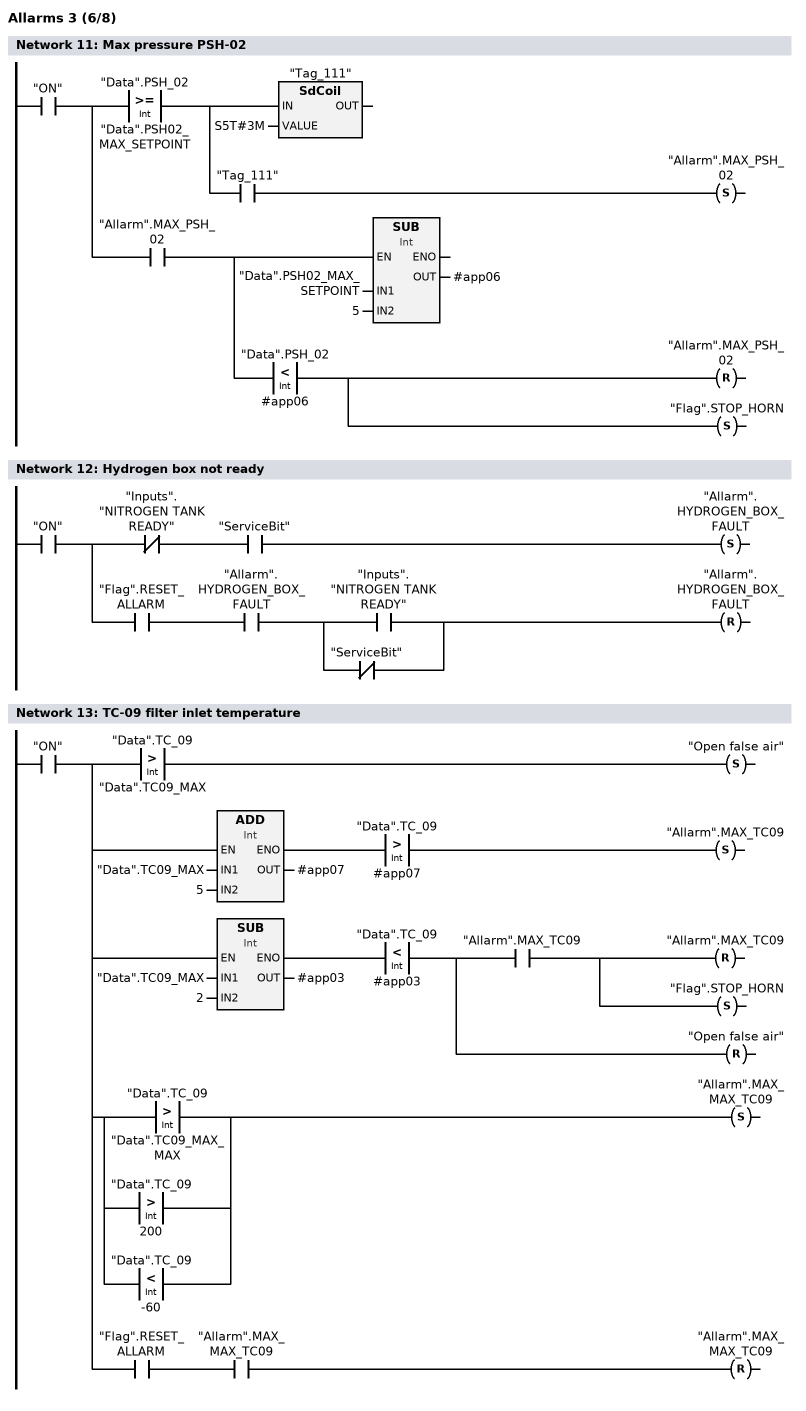
   // no SCL statement known for SdCoil: written as a call
   #_w1 := "ON" AND ("Data".PSH_02 >= "Data".PSH02_MAX_SETPOINT);
   #_w2 := "ON";
   SdCoil(in := #_w1, value := S5T#3M, operand := "Tag_111");
   IF #_w1 AND "Tag_111" THEN "Allarm".MAX_PSH_02 := TRUE; END_IF;
   #_w3 := #_w2 AND "Allarm".MAX_PSH_02;
   IF #_w3 THEN #app06 := "Data".PSH02_MAX_SETPOINT - 5; END_IF;
   IF #_w3 AND ("Data".PSH_02 < #app06) THEN
       "Allarm".MAX_PSH_02 := FALSE;
       "Flag".STOP_HORN := TRUE;
   END_IF;
END_REGION

REGION Network 12: Hydrogen box not ready
   RUNG wire#powerrail
      Contact( "ON" )
      wire#w1
      I_Contact( "Inputs"."NITROGEN TANK READY" )
      Contact( "ServiceBit" )
      S_Coil( "Allarm".HYDROGEN_BOX_FAULT )
   END_RUNG
   RUNG wire#w1
      Contact( "Flag".RESET_ALLARM )
      Contact( "Allarm".HYDROGEN_BOX_FAULT )
      wire#w2
      Contact( "Inputs"."NITROGEN TANK READY" )
      wire#w3
      R_Coil( "Allarm".HYDROGEN_BOX_FAULT )
   END_RUNG
   RUNG wire#w2
      I_Contact( "ServiceBit" )
   END_RUNG wire#w3
   // the same network as SCL:
   IF "ON" AND NOT "Inputs"."NITROGEN TANK READY" AND "ServiceBit" THEN
       "Allarm".HYDROGEN_BOX_FAULT := TRUE;
   END_IF;
   IF "ON" AND "Flag".RESET_ALLARM AND "Allarm".HYDROGEN_BOX_FAULT AND ("Inputs"."NITROGEN TANK READY" OR NOT "ServiceBit") THEN
       "Allarm".HYDROGEN_BOX_FAULT := FALSE;
   END_IF;
END_REGION

REGION Network 13: TC-09 filter inlet temperature
   RUNG wire#powerrail
      Contact( "ON" )
      wire#w1
      { S7_Templates := "SrcType := Int" } GT_Contact(in1 := "Data".TC_09, in2 := "Data".TC09_MAX)
      S_Coil( "Open false air" )
   END_RUNG
   RUNG wire#w1
      { S7_Templates := "SrcType := Int"; S7_GenerateENO := "TRUE" } Add(in1 := "Data".TC09_MAX, in2 := 5, out => #app07)
      { S7_Templates := "SrcType := Int" } GT_Contact(in1 := "Data".TC_09, in2 := #app07)
      S_Coil( "Allarm".MAX_TC09 )
   END_RUNG
   RUNG wire#w1
      { S7_Templates := "SrcType := Int"; S7_GenerateENO := "TRUE" } Sub(in1 := "Data".TC09_MAX, in2 := 2, out => #app03)
      { S7_Templates := "SrcType := Int" } LT_Contact(in1 := "Data".TC_09, in2 := #app03)
      wire#w2
      Contact( "Allarm".MAX_TC09 )
      wire#w3
      R_Coil( "Allarm".MAX_TC09 )
   END_RUNG
   RUNG wire#w3
      S_Coil( "Flag".STOP_HORN )
   END_RUNG
   RUNG wire#w2
      R_Coil( "Open false air" )
   END_RUNG
   RUNG wire#w1
      { S7_Templates := "SrcType := Int" } GT_Contact(in1 := "Data".TC_09, in2 := "Data".TC09_MAX_MAX)
      wire#w4
      S_Coil( "Allarm".MAX_MAX_TC09 )
   END_RUNG
   RUNG wire#w1
      { S7_Templates := "SrcType := Int" } GT_Contact(in1 := "Data".TC_09, in2 := 200)
   END_RUNG wire#w4
   RUNG wire#w1
      { S7_Templates := "SrcType := Int" } LT_Contact(in1 := "Data".TC_09, in2 := -60)
   END_RUNG wire#w4
   RUNG wire#w1
      Contact( "Flag".RESET_ALLARM )
      Contact( "Allarm".MAX_MAX_TC09 )
      R_Coil( "Allarm".MAX_MAX_TC09 )
   END_RUNG
   // the same network as SCL:
   // ENO of a box is taken as its EN; it also drops when the box reports an error
   IF "ON" AND ("Data".TC_09 > "Data".TC09_MAX) THEN "Open false air" := TRUE; END_IF;
   IF "ON" THEN #app07 := "Data".TC09_MAX + 5; END_IF;
   IF "ON" AND ("Data".TC_09 > #app07) THEN "Allarm".MAX_TC09 := TRUE; END_IF;
   IF "ON" THEN #app03 := "Data".TC09_MAX - 2; END_IF;
   #_w1 := "ON" AND ("Data".TC_09 < #app03);
   #_w2 := #_w1 AND "Allarm".MAX_TC09;
   IF #_w2 THEN
       "Allarm".MAX_TC09 := FALSE;
       "Flag".STOP_HORN := TRUE;
   END_IF;
   IF #_w1 THEN "Open false air" := FALSE; END_IF;
   IF "ON" AND (("Data".TC_09 > "Data".TC09_MAX_MAX) OR ("Data".TC_09 > 200) OR ("Data".TC_09 < (-60))) THEN
       "Allarm".MAX_MAX_TC09 := TRUE;
   END_IF;
   IF "ON" AND "Flag".RESET_ALLARM AND "Allarm".MAX_MAX_TC09 THEN "Allarm".MAX_MAX_TC09 := FALSE; END_IF;
END_REGION

REGION Network 14: Max filter depressure
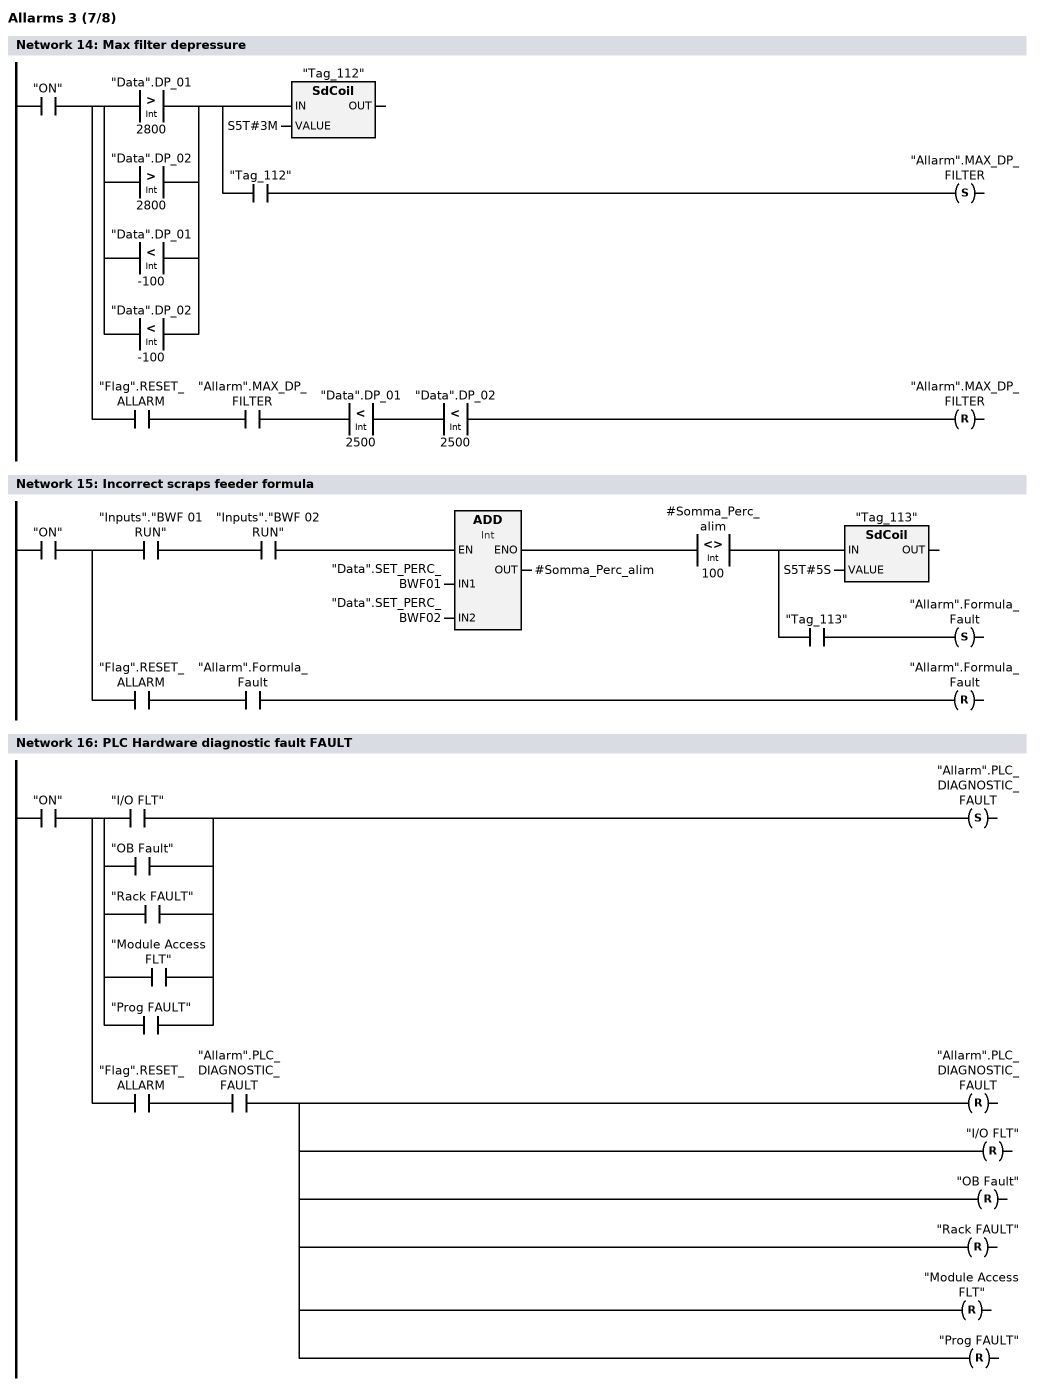
   // no SCL statement known for SdCoil: written as a call
   #_w1 := "ON" AND (("Data".DP_01 > 2800) OR ("Data".DP_02 > 2800) OR ("Data".DP_01 < (-100)) OR ("Data".DP_02 < (-100)));
   #_w2 := "ON";
   SdCoil(in := #_w1, value := S5T#3M, operand := "Tag_112");
   IF #_w1 AND "Tag_112" THEN "Allarm".MAX_DP_FILTER := TRUE; END_IF;
   IF #_w2 AND "Flag".RESET_ALLARM AND "Allarm".MAX_DP_FILTER AND ("Data".DP_01 < 2500) AND ("Data".DP_02 < 2500) THEN
       "Allarm".MAX_DP_FILTER := FALSE;
   END_IF;
END_REGION

REGION Network 15: Incorrect scraps feeder formula
   // no SCL statement known for SdCoil: written as a call
   // ENO of a box is taken as its EN; it also drops when the box reports an error
   #_w1 := "ON" AND "Inputs"."BWF 01 RUN" AND "Inputs"."BWF 02 RUN";
   IF #_w1 THEN #Somma_Perc_alim := "Data".SET_PERC_BWF01 + "Data".SET_PERC_BWF02; END_IF;
   #_w2 := #_w1 AND (#Somma_Perc_alim <> 100);
   #_w3 := "ON";
   SdCoil(in := #_w2, value := S5T#5S, operand := "Tag_113");
   IF #_w2 AND "Tag_113" THEN "Allarm".Formula_Fault := TRUE; END_IF;
   IF #_w3 AND "Flag".RESET_ALLARM AND "Allarm".Formula_Fault THEN "Allarm".Formula_Fault := FALSE; END_IF;
END_REGION

REGION Network 16: PLC Hardware diagnostic fault FAULT
   RUNG wire#powerrail
      Contact( "ON" )
      wire#w1
      Contact( "I/O FLT" )
      wire#w2
      S_Coil( "Allarm".PLC_DIAGNOSTIC_FAULT )
   END_RUNG
   RUNG wire#w1
      Contact( "OB Fault" )
   END_RUNG wire#w2
   RUNG wire#w1
      Contact( "Rack FAULT" )
   END_RUNG wire#w2
   RUNG wire#w1
      Contact( "Module Access FLT" )
   END_RUNG wire#w2
   RUNG wire#w1
      Contact( "Prog FAULT" )
   END_RUNG wire#w2
   RUNG wire#w1
      Contact( "Flag".RESET_ALLARM )
      Contact( "Allarm".PLC_DIAGNOSTIC_FAULT )
      wire#w3
      R_Coil( "Allarm".PLC_DIAGNOSTIC_FAULT )
   END_RUNG
   RUNG wire#w3
      R_Coil( "I/O FLT" )
   END_RUNG
   RUNG wire#w3
      R_Coil( "OB Fault" )
   END_RUNG
   RUNG wire#w3
      R_Coil( "Rack FAULT" )
   END_RUNG
   RUNG wire#w3
      R_Coil( "Module Access FLT" )
   END_RUNG
   RUNG wire#w3
      R_Coil( "Prog FAULT" )
   END_RUNG
   // the same network as SCL:
   IF "ON" AND ("I/O FLT" OR "OB Fault" OR "Rack FAULT" OR "Module Access FLT" OR "Prog FAULT") THEN
       "Allarm".PLC_DIAGNOSTIC_FAULT := TRUE;
   END_IF;
   #_w1 := "ON" AND "Flag".RESET_ALLARM AND "Allarm".PLC_DIAGNOSTIC_FAULT;
   IF #_w1 THEN
       "Allarm".PLC_DIAGNOSTIC_FAULT := FALSE;
       "I/O FLT" := FALSE;
       "OB Fault" := FALSE;
       "Rack FAULT" := FALSE;
       "Module Access FLT" := FALSE;
       "Prog FAULT" := FALSE;
   END_IF;
END_REGION

REGION Network 17: Ro03
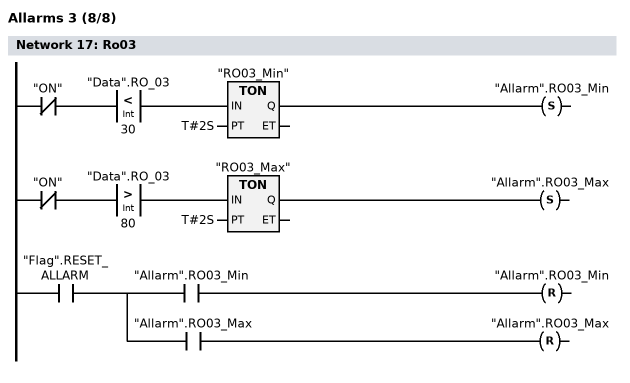
   "RO03_Min".TON(IN := NOT "ON" AND ("Data".RO_03 < 30), PT := T#2S);
   IF "RO03_Min".Q THEN "Allarm".RO03_Min := TRUE; END_IF;
   "RO03_Max".TON(IN := NOT "ON" AND ("Data".RO_03 > 80), PT := T#2S);
   IF "RO03_Max".Q THEN "Allarm".RO03_Max := TRUE; END_IF;
   IF "Flag".RESET_ALLARM AND "Allarm".RO03_Min THEN "Allarm".RO03_Min := FALSE; END_IF;
   IF "Flag".RESET_ALLARM AND "Allarm".RO03_Max THEN "Allarm".RO03_Max := FALSE; END_IF;
END_REGION
END_FUNCTION

FUNCTION "Motors 1" : Void   // FC7, LAD
{ S7_Optimized_Access := 'FALSE' }
VERSION : 0.1
   VAR_TEMP
      Start_LD01Vib : Bool;
      Disable_Load_RD01 : Bool;
      Stop_Fan_FN01 : Bool;
      Stop_Fan_FN04 : Bool;
      TimConv : Word;
   END_VAR
   VAR_TEMP   // added for the SCL form of the ladder/FBD networks
      _w1 : Bool;
      _w2 : Bool;
      _w3 : Bool;
   END_VAR
BEGIN

REGION Network 1: Enable maintenance mode / MAINTENANCE
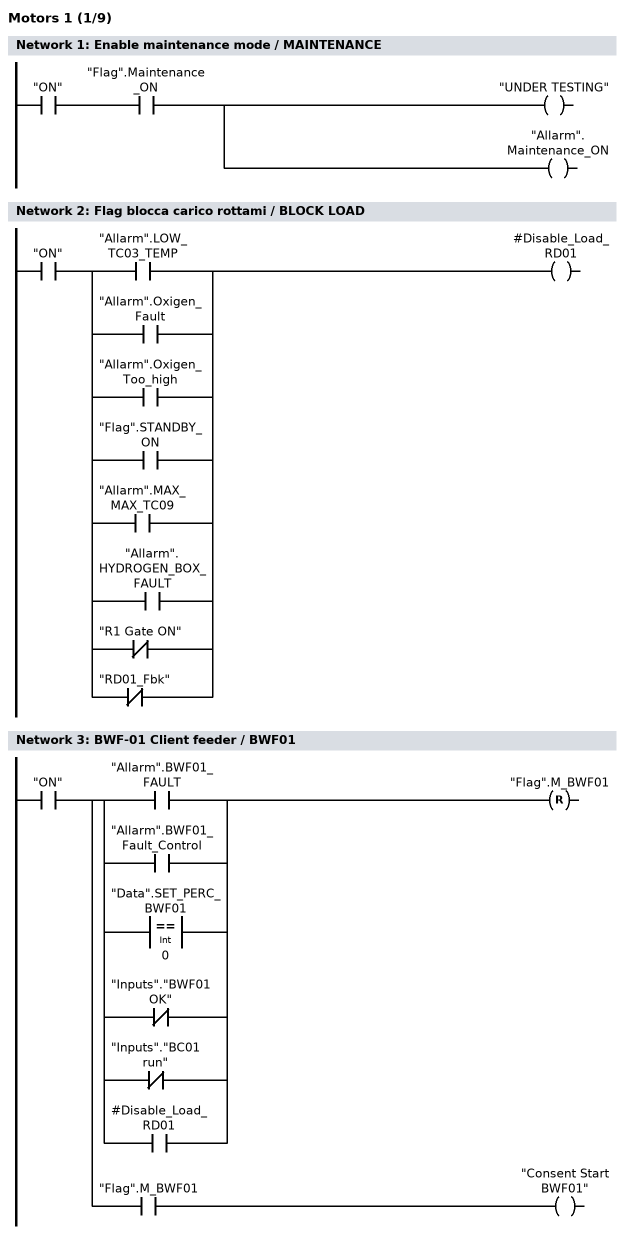
   RUNG wire#powerrail
      Contact( "ON" )
      Contact( "Flag".Maintenance_ON )
      wire#w1
      Coil( "UNDER TESTING" )
   END_RUNG
   RUNG wire#w1
      Coil( "Allarm".Maintenance_ON )
   END_RUNG
   // the same network as SCL:
   "UNDER TESTING" := "ON" AND "Flag".Maintenance_ON;
   "Allarm".Maintenance_ON := "UNDER TESTING";
END_REGION

REGION Network 2: Flag blocca carico rottami / BLOCK LOAD
   RUNG wire#powerrail
      Contact( "ON" )
      wire#w1
      Contact( "Allarm".LOW_TC03_TEMP )
      wire#w2
      Coil( #Disable_Load_RD01 )
   END_RUNG
   RUNG wire#w1
      Contact( "Allarm".Oxigen_Fault )
   END_RUNG wire#w2
   RUNG wire#w1
      Contact( "Allarm".Oxigen_Too_high )
   END_RUNG wire#w2
   RUNG wire#w1
      Contact( "Flag".STANDBY_ON )
   END_RUNG wire#w2
   RUNG wire#w1
      Contact( "Allarm".MAX_MAX_TC09 )
   END_RUNG wire#w2
   RUNG wire#w1
      Contact( "Allarm".HYDROGEN_BOX_FAULT )
   END_RUNG wire#w2
   RUNG wire#w1
      I_Contact( "R1 Gate ON" )
   END_RUNG wire#w2
   RUNG wire#w1
      I_Contact( "RD01_Fbk" )
   END_RUNG wire#w2
   // the same network as SCL:
   #Disable_Load_RD01 := "ON" AND ("Allarm".LOW_TC03_TEMP OR "Allarm".Oxigen_Fault OR "Allarm".Oxigen_Too_high OR "Flag".STANDBY_ON OR "Allarm".MAX_MAX_TC09 OR "Allarm".HYDROGEN_BOX_FAULT OR NOT "R1 Gate ON" OR NOT "RD01_Fbk");
END_REGION

REGION Network 3: BWF-01 Client feeder / BWF01
   RUNG wire#powerrail
      Contact( "ON" )
      wire#w1
      Contact( "Allarm".BWF01_FAULT )
      wire#w2
      R_Coil( "Flag".M_BWF01 )
   END_RUNG
   RUNG wire#w1
      Contact( "Allarm".BWF01_Fault_Control )
   END_RUNG wire#w2
   RUNG wire#w1
      { S7_Templates := "SrcType := Int" } EQ_Contact(in1 := "Data".SET_PERC_BWF01, in2 := 0)
   END_RUNG wire#w2
   RUNG wire#w1
      I_Contact( "Inputs"."BWF01 OK" )
   END_RUNG wire#w2
   RUNG wire#w1
      I_Contact( "Inputs"."BC01 run" )
   END_RUNG wire#w2
   RUNG wire#w1
      Contact( #Disable_Load_RD01 )
   END_RUNG wire#w2
   RUNG wire#w1
      Contact( "Flag".M_BWF01 )
      Coil( "Consent Start BWF01" )
   END_RUNG
   // the same network as SCL:
   IF "ON" AND ("Allarm".BWF01_FAULT OR "Allarm".BWF01_Fault_Control OR ("Data".SET_PERC_BWF01 = 0) OR NOT "Inputs"."BWF01 OK" OR NOT "Inputs"."BC01 run" OR #Disable_Load_RD01) THEN
       "Flag".M_BWF01 := FALSE;
   END_IF;
   "Consent Start BWF01" := "ON" AND "Flag".M_BWF01;
END_REGION

REGION Network 4: BWF-02 Client feeder / BWF02
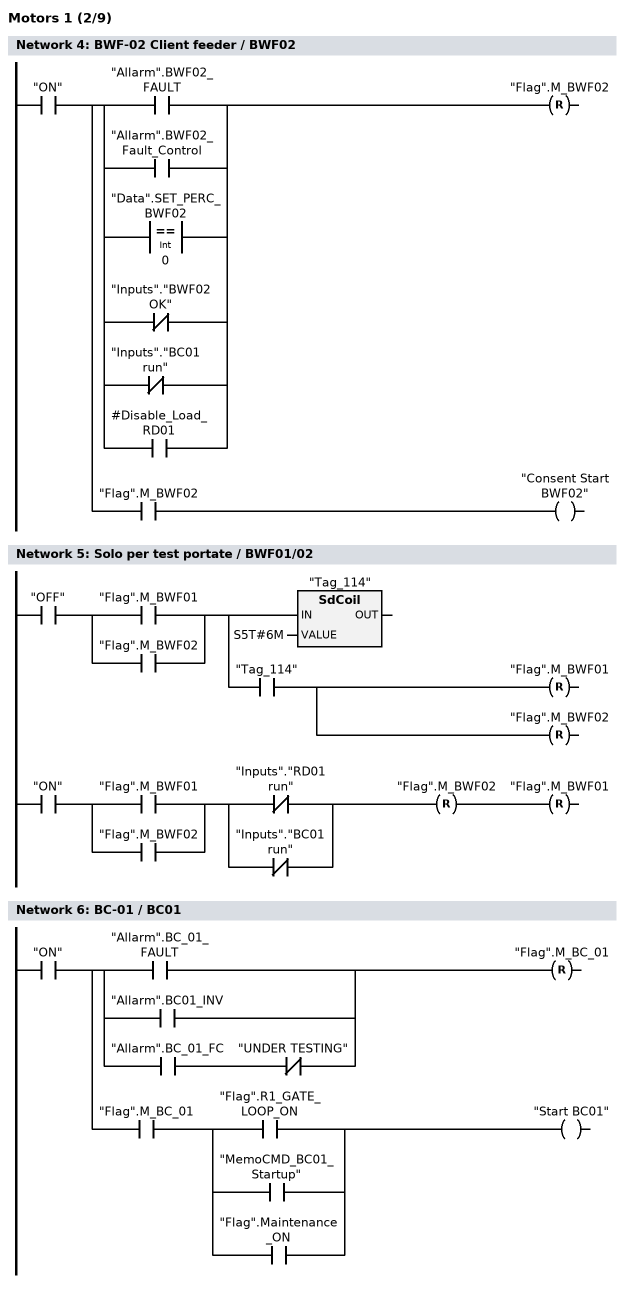
   RUNG wire#powerrail
      Contact( "ON" )
      wire#w1
      Contact( "Allarm".BWF02_FAULT )
      wire#w2
      R_Coil( "Flag".M_BWF02 )
   END_RUNG
   RUNG wire#w1
      Contact( "Allarm".BWF02_Fault_Control )
   END_RUNG wire#w2
   RUNG wire#w1
      { S7_Templates := "SrcType := Int" } EQ_Contact(in1 := "Data".SET_PERC_BWF02, in2 := 0)
   END_RUNG wire#w2
   RUNG wire#w1
      I_Contact( "Inputs"."BWF02 OK" )
   END_RUNG wire#w2
   RUNG wire#w1
      I_Contact( "Inputs"."BC01 run" )
   END_RUNG wire#w2
   RUNG wire#w1
      Contact( #Disable_Load_RD01 )
   END_RUNG wire#w2
   RUNG wire#w1
      Contact( "Flag".M_BWF02 )
      Coil( "Consent Start BWF02" )
   END_RUNG
   // the same network as SCL:
   IF "ON" AND ("Allarm".BWF02_FAULT OR "Allarm".BWF02_Fault_Control OR ("Data".SET_PERC_BWF02 = 0) OR NOT "Inputs"."BWF02 OK" OR NOT "Inputs"."BC01 run" OR #Disable_Load_RD01) THEN
       "Flag".M_BWF02 := FALSE;
   END_IF;
   "Consent Start BWF02" := "ON" AND "Flag".M_BWF02;
END_REGION

REGION Network 5: Solo per test portate / BWF01/02
   // no SCL statement known for SdCoil: written as a call
   #_w1 := "OFF" AND ("Flag".M_BWF01 OR "Flag".M_BWF02);
   SdCoil(in := #_w1, value := S5T#6M, operand := "Tag_114");
   IF #_w1 AND "Tag_114" THEN
       "Flag".M_BWF01 := FALSE;
       "Flag".M_BWF02 := FALSE;
   END_IF;
   #_w2 := "ON" AND ("Flag".M_BWF01 OR "Flag".M_BWF02) AND (NOT "Inputs"."RD01 run" OR NOT "Inputs"."BC01 run");
   IF #_w2 THEN
       "Flag".M_BWF02 := FALSE;
       "Flag".M_BWF01 := FALSE;
   END_IF;
END_REGION

REGION Network 6: BC-01 / BC01
   RUNG wire#powerrail
      Contact( "ON" )
      wire#w1
      Contact( "Allarm".BC_01_FAULT )
      wire#w2
      R_Coil( "Flag".M_BC_01 )
   END_RUNG
   RUNG wire#w1
      Contact( "Allarm".BC01_INV )
   END_RUNG wire#w2
   RUNG wire#w1
      Contact( "Allarm".BC_01_FC )
      I_Contact( "UNDER TESTING" )
   END_RUNG wire#w2
   RUNG wire#w1
      Contact( "Flag".M_BC_01 )
      wire#w3
      Contact( "Flag".R1_GATE_LOOP_ON )
      wire#w4
      Coil( "Start BC01" )
   END_RUNG
   RUNG wire#w3
      Contact( "MemoCMD_BC01_Startup" )
   END_RUNG wire#w4
   RUNG wire#w3
      Contact( "Flag".Maintenance_ON )
   END_RUNG wire#w4
   // the same network as SCL:
   IF "ON" AND ("Allarm".BC_01_FAULT OR "Allarm".BC01_INV OR ("Allarm".BC_01_FC AND NOT "UNDER TESTING")) THEN
       "Flag".M_BC_01 := FALSE;
   END_IF;
   "Start BC01" := "ON" AND "Flag".M_BC_01 AND ("Flag".R1_GATE_LOOP_ON OR "MemoCMD_BC01_Startup" OR "Flag".Maintenance_ON);
END_REGION

REGION Network 7: RD-01 / RD01
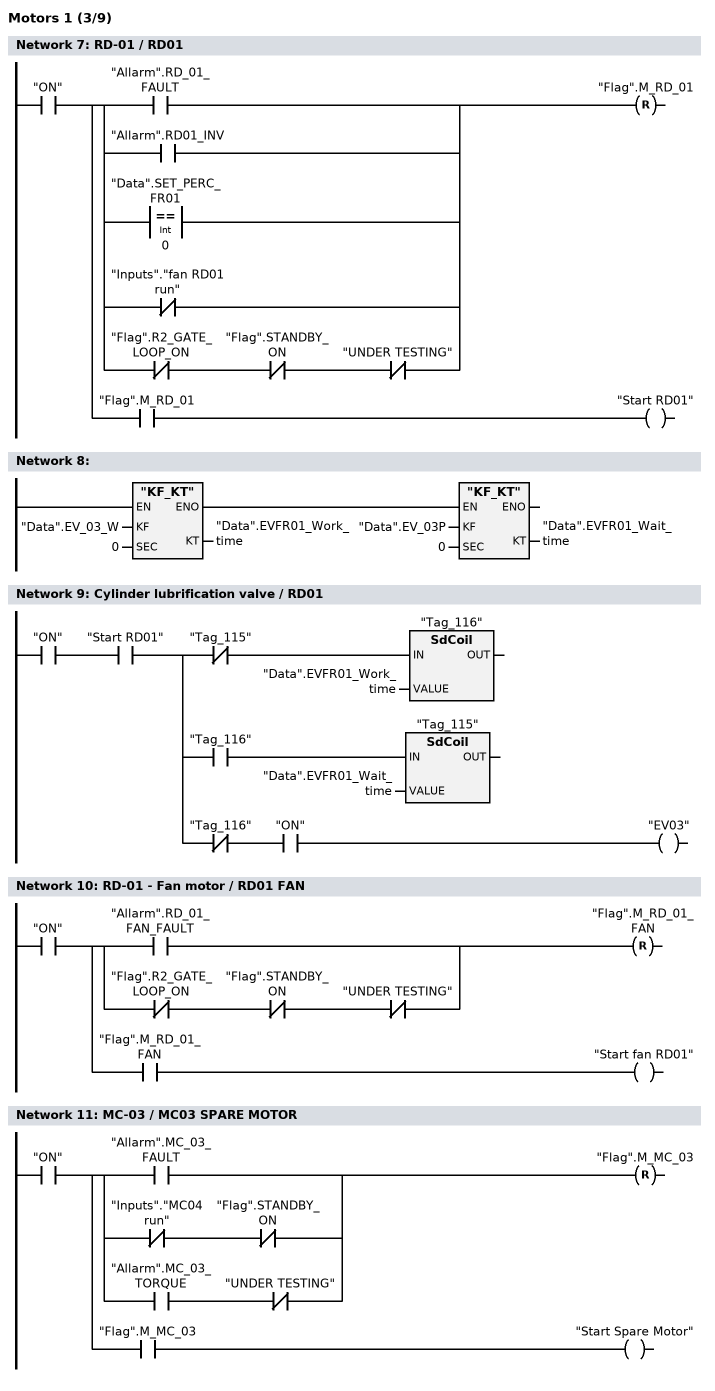
   RUNG wire#powerrail
      Contact( "ON" )
      wire#w1
      Contact( "Allarm".RD_01_FAULT )
      wire#w2
      R_Coil( "Flag".M_RD_01 )
   END_RUNG
   RUNG wire#w1
      Contact( "Allarm".RD01_INV )
   END_RUNG wire#w2
   RUNG wire#w1
      { S7_Templates := "SrcType := Int" } EQ_Contact(in1 := "Data".SET_PERC_FR01, in2 := 0)
   END_RUNG wire#w2
   RUNG wire#w1
      I_Contact( "Inputs"."fan RD01 run" )
   END_RUNG wire#w2
   RUNG wire#w1
      I_Contact( "Flag".R2_GATE_LOOP_ON )
      I_Contact( "Flag".STANDBY_ON )
      I_Contact( "UNDER TESTING" )
   END_RUNG wire#w2
   RUNG wire#w1
      Contact( "Flag".M_RD_01 )
      Coil( "Start RD01" )
   END_RUNG
   // the same network as SCL:
   IF "ON" AND ("Allarm".RD_01_FAULT OR "Allarm".RD01_INV OR ("Data".SET_PERC_FR01 = 0) OR NOT "Inputs"."fan RD01 run" OR (NOT "Flag".R2_GATE_LOOP_ON AND NOT "Flag".STANDBY_ON AND NOT "UNDER TESTING")) THEN
       "Flag".M_RD_01 := FALSE;
   END_IF;
   "Start RD01" := "ON" AND "Flag".M_RD_01;
END_REGION

REGION Network 8
   RUNG wire#powerrail
      "KF_KT"(KF := "Data".EV_03_W, SEC := 0, KT => "Data".EVFR01_Work_time)
      "KF_KT"(KF := "Data".EV_03P, SEC := 0, KT => "Data".EVFR01_Wait_time)
   END_RUNG
   // the same network as SCL:
   "KF_KT"(KF := "Data".EV_03_W, SEC := 0, KT => "Data".EVFR01_Work_time, ENO => #_w1);
   IF #_w1 THEN "KF_KT"(KF := "Data".EV_03P, SEC := 0, KT => "Data".EVFR01_Wait_time); END_IF;
END_REGION

REGION Network 9: Cylinder lubrification valve / RD01
   // no SCL statement known for SdCoil: written as a call
   #_w1 := "ON" AND "Start RD01";
   SdCoil(in := #_w1 AND NOT "Tag_115", value := "Data".EVFR01_Work_time, operand := "Tag_116");
   SdCoil(in := #_w1 AND "Tag_116", value := "Data".EVFR01_Wait_time, operand := "Tag_115");
   "EV03" := #_w1 AND NOT "Tag_116" AND "ON";
END_REGION

REGION Network 10: RD-01 - Fan motor / RD01 FAN
   RUNG wire#powerrail
      Contact( "ON" )
      wire#w1
      Contact( "Allarm".RD_01_FAN_FAULT )
      wire#w2
      R_Coil( "Flag".M_RD_01_FAN )
   END_RUNG
   RUNG wire#w1
      I_Contact( "Flag".R2_GATE_LOOP_ON )
      I_Contact( "Flag".STANDBY_ON )
      I_Contact( "UNDER TESTING" )
   END_RUNG wire#w2
   RUNG wire#w1
      Contact( "Flag".M_RD_01_FAN )
      Coil( "Start fan RD01" )
   END_RUNG
   // the same network as SCL:
   IF "ON" AND ("Allarm".RD_01_FAN_FAULT OR (NOT "Flag".R2_GATE_LOOP_ON AND NOT "Flag".STANDBY_ON AND NOT "UNDER TESTING")) THEN
       "Flag".M_RD_01_FAN := FALSE;
   END_IF;
   "Start fan RD01" := "ON" AND "Flag".M_RD_01_FAN;
END_REGION

REGION Network 11: MC-03 / MC03 SPARE MOTOR
   RUNG wire#powerrail
      Contact( "ON" )
      wire#w1
      Contact( "Allarm".MC_03_FAULT )
      wire#w2
      R_Coil( "Flag".M_MC_03 )
   END_RUNG
   RUNG wire#w1
      I_Contact( "Inputs"."MC04 run" )
      I_Contact( "Flag".STANDBY_ON )
   END_RUNG wire#w2
   RUNG wire#w1
      Contact( "Allarm".MC_03_TORQUE )
      I_Contact( "UNDER TESTING" )
   END_RUNG wire#w2
   RUNG wire#w1
      Contact( "Flag".M_MC_03 )
      Coil( "Start Spare Motor" )
   END_RUNG
   // the same network as SCL:
   IF "ON" AND ("Allarm".MC_03_FAULT OR (NOT "Inputs"."MC04 run" AND NOT "Flag".STANDBY_ON) OR ("Allarm".MC_03_TORQUE AND NOT "UNDER TESTING")) THEN
       "Flag".M_MC_03 := FALSE;
   END_IF;
   "Start Spare Motor" := "ON" AND "Flag".M_MC_03;
END_REGION

REGION Network 12: MC-04 / MC04
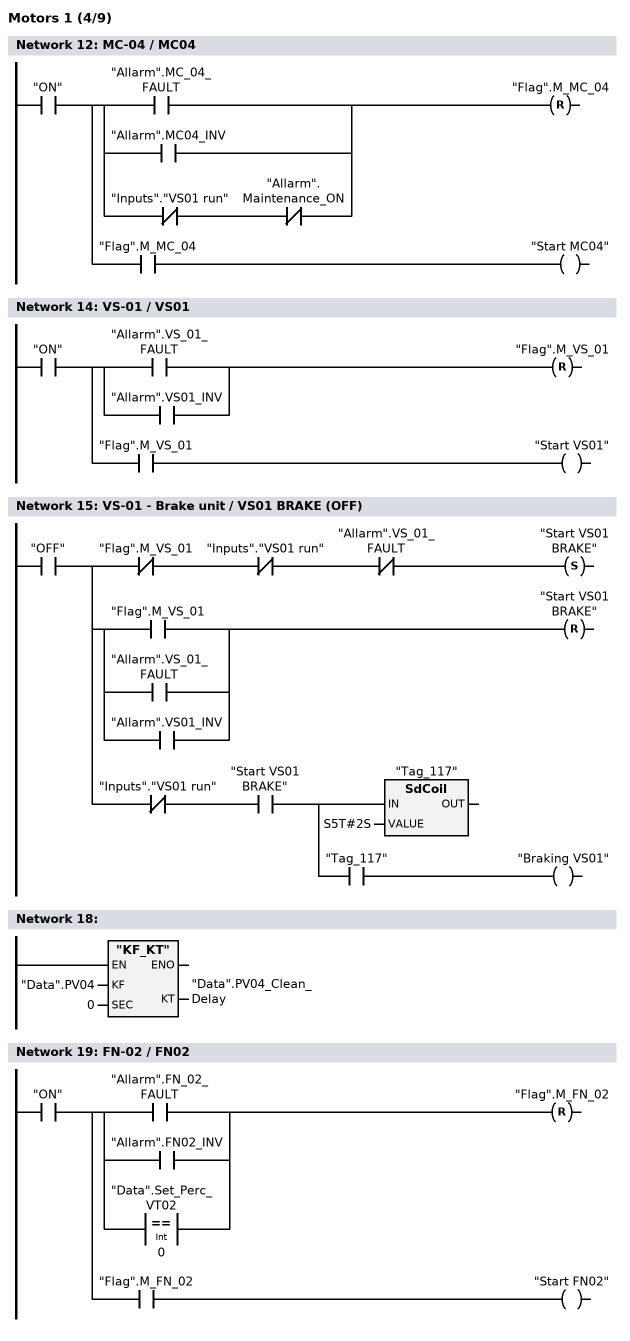
   RUNG wire#powerrail
      Contact( "ON" )
      wire#w1
      Contact( "Allarm".MC_04_FAULT )
      wire#w2
      R_Coil( "Flag".M_MC_04 )
   END_RUNG
   RUNG wire#w1
      Contact( "Allarm".MC04_INV )
   END_RUNG wire#w2
   RUNG wire#w1
      I_Contact( "Inputs"."VS01 run" )
      I_Contact( "Allarm".Maintenance_ON )
   END_RUNG wire#w2
   RUNG wire#w1
      Contact( "Flag".M_MC_04 )
      Coil( "Start MC04" )
   END_RUNG
   // the same network as SCL:
   IF "ON" AND ("Allarm".MC_04_FAULT OR "Allarm".MC04_INV OR (NOT "Inputs"."VS01 run" AND NOT "Allarm".Maintenance_ON)) THEN
       "Flag".M_MC_04 := FALSE;
   END_IF;
   "Start MC04" := "ON" AND "Flag".M_MC_04;
END_REGION

REGION Network 13: MC-05 / MC05 DELETED
END_REGION

REGION Network 14: VS-01 / VS01
   RUNG wire#powerrail
      Contact( "ON" )
      wire#w1
      Contact( "Allarm".VS_01_FAULT )
      wire#w2
      R_Coil( "Flag".M_VS_01 )
   END_RUNG
   RUNG wire#w1
      Contact( "Allarm".VS01_INV )
   END_RUNG wire#w2
   RUNG wire#w1
      Contact( "Flag".M_VS_01 )
      Coil( "Start VS01" )
   END_RUNG
   // the same network as SCL:
   IF "ON" AND ("Allarm".VS_01_FAULT OR "Allarm".VS01_INV) THEN "Flag".M_VS_01 := FALSE; END_IF;
   "Start VS01" := "ON" AND "Flag".M_VS_01;
END_REGION

REGION Network 15: VS-01 - Brake unit / VS01 BRAKE (OFF)
   // no SCL statement known for SdCoil: written as a call
   IF "OFF" AND NOT "Flag".M_VS_01 AND NOT "Inputs"."VS01 run" AND NOT "Allarm".VS_01_FAULT THEN
       "Start VS01 BRAKE" := TRUE;
   END_IF;
   IF "OFF" AND ("Flag".M_VS_01 OR "Allarm".VS_01_FAULT OR "Allarm".VS01_INV) THEN
       "Start VS01 BRAKE" := FALSE;
   END_IF;
   #_w1 := "OFF" AND NOT "Inputs"."VS01 run" AND "Start VS01 BRAKE";
   SdCoil(in := #_w1, value := S5T#2S, operand := "Tag_117");
   "Braking VS01" := #_w1 AND "Tag_117";
END_REGION

REGION Network 16: SC-12 screw discharge drum dust / SC12 DELETED
END_REGION

REGION Network 17: Valve discharge drum dust / PV04 DELETED
END_REGION

REGION Network 18
   RUNG wire#powerrail
      "KF_KT"(KF := "Data".PV04, SEC := 0, KT => "Data".PV04_Clean_Delay)
   END_RUNG
   // the same network as SCL:
   "KF_KT"(KF := "Data".PV04, SEC := 0, KT => "Data".PV04_Clean_Delay);
END_REGION

REGION Network 19: FN-02 / FN02
   RUNG wire#powerrail
      Contact( "ON" )
      wire#w1
      Contact( "Allarm".FN_02_FAULT )
      wire#w2
      R_Coil( "Flag".M_FN_02 )
   END_RUNG
   RUNG wire#w1
      Contact( "Allarm".FN02_INV )
   END_RUNG wire#w2
   RUNG wire#w1
      { S7_Templates := "SrcType := Int" } EQ_Contact(in1 := "Data".Set_Perc_VT02, in2 := 0)
   END_RUNG wire#w2
   RUNG wire#w1
      Contact( "Flag".M_FN_02 )
      Coil( "Start FN02" )
   END_RUNG
   // the same network as SCL:
   IF "ON" AND ("Allarm".FN_02_FAULT OR "Allarm".FN02_INV OR ("Data".Set_Perc_VT02 = 0)) THEN
       "Flag".M_FN_02 := FALSE;
   END_IF;
   "Start FN02" := "ON" AND "Flag".M_FN_02;
END_REGION

REGION Network 20: VR-01 / VR01
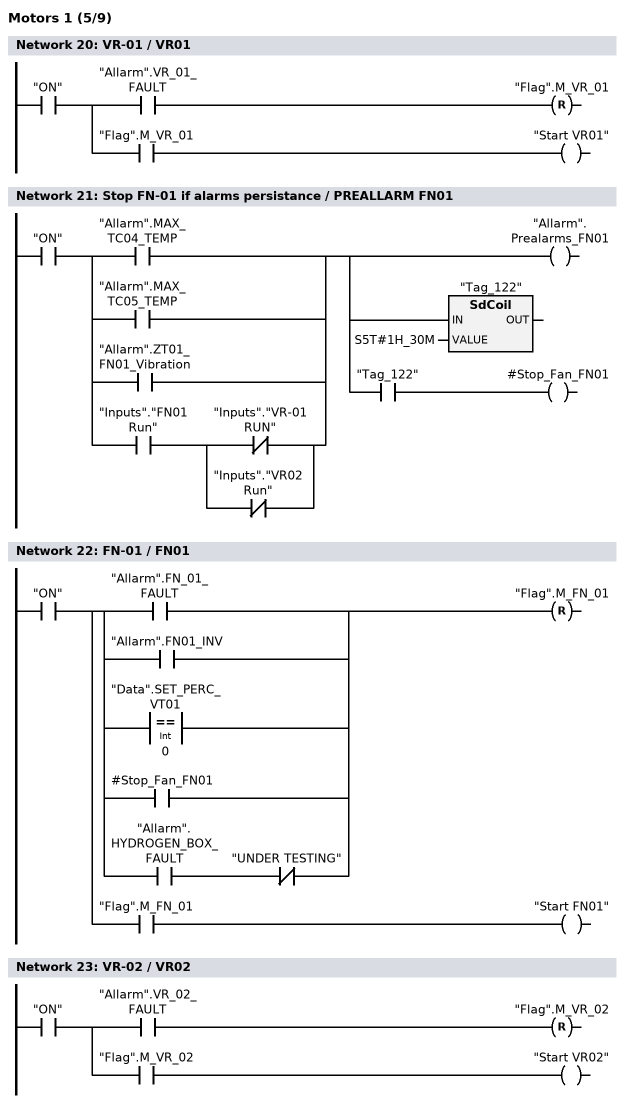
   RUNG wire#powerrail
      Contact( "ON" )
      wire#w1
      Contact( "Allarm".VR_01_FAULT )
      R_Coil( "Flag".M_VR_01 )
   END_RUNG
   RUNG wire#w1
      Contact( "Flag".M_VR_01 )
      Coil( "Start VR01" )
   END_RUNG
   // the same network as SCL:
   IF "ON" AND "Allarm".VR_01_FAULT THEN "Flag".M_VR_01 := FALSE; END_IF;
   "Start VR01" := "ON" AND "Flag".M_VR_01;
END_REGION

REGION Network 21: Stop FN-01 if alarms persistance / PREALLARM FN01
   // no SCL statement known for SdCoil: written as a call
   "Allarm".Prealarms_FN01 := "ON" AND ("Allarm".MAX_TC04_TEMP OR "Allarm".MAX_TC05_TEMP OR "Allarm".ZT01_FN01_Vibration OR ("Inputs"."FN01 Run" AND (NOT "Inputs"."VR-01 RUN" OR NOT "Inputs"."VR02 Run")));
   #_w1 := "Allarm".Prealarms_FN01;
   SdCoil(in := "Allarm".Prealarms_FN01, value := S5T#1H_30M, operand := "Tag_122");
   #Stop_Fan_FN01 := #_w1 AND "Tag_122";
END_REGION

REGION Network 22: FN-01 / FN01
   RUNG wire#powerrail
      Contact( "ON" )
      wire#w1
      Contact( "Allarm".FN_01_FAULT )
      wire#w2
      R_Coil( "Flag".M_FN_01 )
   END_RUNG
   RUNG wire#w1
      Contact( "Allarm".FN01_INV )
   END_RUNG wire#w2
   RUNG wire#w1
      { S7_Templates := "SrcType := Int" } EQ_Contact(in1 := "Data".SET_PERC_VT01, in2 := 0)
   END_RUNG wire#w2
   RUNG wire#w1
      Contact( #Stop_Fan_FN01 )
   END_RUNG wire#w2
   RUNG wire#w1
      Contact( "Allarm".HYDROGEN_BOX_FAULT )
      I_Contact( "UNDER TESTING" )
   END_RUNG wire#w2
   RUNG wire#w1
      Contact( "Flag".M_FN_01 )
      Coil( "Start FN01" )
   END_RUNG
   // the same network as SCL:
   IF "ON" AND ("Allarm".FN_01_FAULT OR "Allarm".FN01_INV OR ("Data".SET_PERC_VT01 = 0) OR #Stop_Fan_FN01 OR ("Allarm".HYDROGEN_BOX_FAULT AND NOT "UNDER TESTING")) THEN
       "Flag".M_FN_01 := FALSE;
   END_IF;
   "Start FN01" := "ON" AND "Flag".M_FN_01;
END_REGION

REGION Network 23: VR-02 / VR02
   RUNG wire#powerrail
      Contact( "ON" )
      wire#w1
      Contact( "Allarm".VR_02_FAULT )
      R_Coil( "Flag".M_VR_02 )
   END_RUNG
   RUNG wire#w1
      Contact( "Flag".M_VR_02 )
      Coil( "Start VR02" )
   END_RUNG
   // the same network as SCL:
   IF "ON" AND "Allarm".VR_02_FAULT THEN "Flag".M_VR_02 := FALSE; END_IF;
   "Start VR02" := "ON" AND "Flag".M_VR_02;
END_REGION

REGION Network 24: CH-01 / CH01
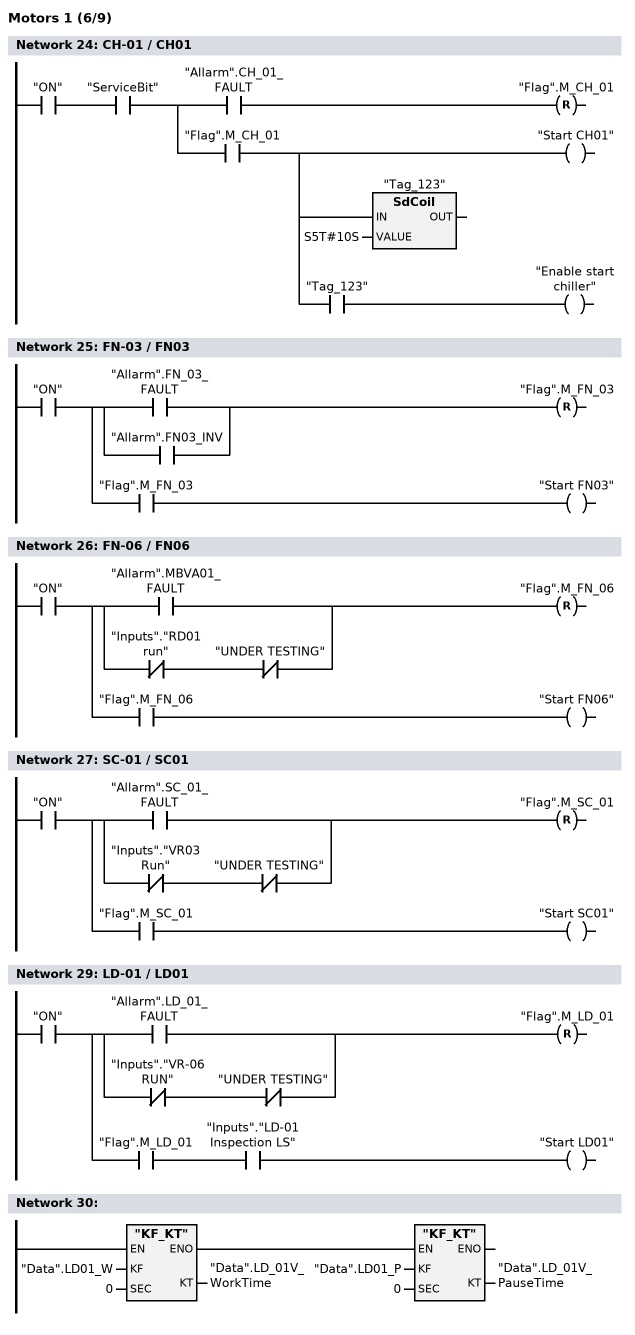
   // no SCL statement known for SdCoil: written as a call
   #_w1 := "ON" AND "ServiceBit";
   IF #_w1 AND "Allarm".CH_01_FAULT THEN "Flag".M_CH_01 := FALSE; END_IF;
   "Start CH01" := #_w1 AND "Flag".M_CH_01;
   #_w2 := "Start CH01";
   SdCoil(in := "Start CH01", value := S5T#10S, operand := "Tag_123");
   "Enable start chiller" := #_w2 AND "Tag_123";
END_REGION

REGION Network 25: FN-03 / FN03
   RUNG wire#powerrail
      Contact( "ON" )
      wire#w1
      Contact( "Allarm".FN_03_FAULT )
      wire#w2
      R_Coil( "Flag".M_FN_03 )
   END_RUNG
   RUNG wire#w1
      Contact( "Allarm".FN03_INV )
   END_RUNG wire#w2
   RUNG wire#w1
      Contact( "Flag".M_FN_03 )
      Coil( "Start FN03" )
   END_RUNG
   // the same network as SCL:
   IF "ON" AND ("Allarm".FN_03_FAULT OR "Allarm".FN03_INV) THEN "Flag".M_FN_03 := FALSE; END_IF;
   "Start FN03" := "ON" AND "Flag".M_FN_03;
END_REGION

REGION Network 26: FN-06 / FN06
   RUNG wire#powerrail
      Contact( "ON" )
      wire#w1
      Contact( "Allarm".MBVA01_FAULT )
      wire#w2
      R_Coil( "Flag".M_FN_06 )
   END_RUNG
   RUNG wire#w1
      I_Contact( "Inputs"."RD01 run" )
      I_Contact( "UNDER TESTING" )
   END_RUNG wire#w2
   RUNG wire#w1
      Contact( "Flag".M_FN_06 )
      Coil( "Start FN06" )
   END_RUNG
   // the same network as SCL:
   IF "ON" AND ("Allarm".MBVA01_FAULT OR (NOT "Inputs"."RD01 run" AND NOT "UNDER TESTING")) THEN
       "Flag".M_FN_06 := FALSE;
   END_IF;
   "Start FN06" := "ON" AND "Flag".M_FN_06;
END_REGION

REGION Network 27: SC-01 / SC01
   RUNG wire#powerrail
      Contact( "ON" )
      wire#w1
      Contact( "Allarm".SC_01_FAULT )
      wire#w2
      R_Coil( "Flag".M_SC_01 )
   END_RUNG
   RUNG wire#w1
      I_Contact( "Inputs"."VR03 Run" )
      I_Contact( "UNDER TESTING" )
   END_RUNG wire#w2
   RUNG wire#w1
      Contact( "Flag".M_SC_01 )
      Coil( "Start SC01" )
   END_RUNG
   // the same network as SCL:
   IF "ON" AND ("Allarm".SC_01_FAULT OR (NOT "Inputs"."VR03 Run" AND NOT "UNDER TESTING")) THEN
       "Flag".M_SC_01 := FALSE;
   END_IF;
   "Start SC01" := "ON" AND "Flag".M_SC_01;
END_REGION

REGION Network 28: FN-01 FAN / FN01 DELETED
END_REGION

REGION Network 29: LD-01 / LD01
   RUNG wire#powerrail
      Contact( "ON" )
      wire#w1
      Contact( "Allarm".LD_01_FAULT )
      wire#w2
      R_Coil( "Flag".M_LD_01 )
   END_RUNG
   RUNG wire#w1
      I_Contact( "Inputs"."VR-06 RUN" )
      I_Contact( "UNDER TESTING" )
   END_RUNG wire#w2
   RUNG wire#w1
      Contact( "Flag".M_LD_01 )
      Contact( "Inputs"."LD-01 Inspection LS" )
      Coil( "Start LD01" )
   END_RUNG
   // the same network as SCL:
   IF "ON" AND ("Allarm".LD_01_FAULT OR (NOT "Inputs"."VR-06 RUN" AND NOT "UNDER TESTING")) THEN
       "Flag".M_LD_01 := FALSE;
   END_IF;
   "Start LD01" := "ON" AND "Flag".M_LD_01 AND "Inputs"."LD-01 Inspection LS";
END_REGION

REGION Network 30
   RUNG wire#powerrail
      "KF_KT"(KF := "Data".LD01_W, SEC := 0, KT => "Data".LD_01V_WorkTime)
      "KF_KT"(KF := "Data".LD01_P, SEC := 0, KT => "Data".LD_01V_PauseTime)
   END_RUNG
   // the same network as SCL:
   "KF_KT"(KF := "Data".LD01_W, SEC := 0, KT => "Data".LD_01V_WorkTime, ENO => #_w1);
   IF #_w1 THEN "KF_KT"(KF := "Data".LD01_P, SEC := 0, KT => "Data".LD_01V_PauseTime); END_IF;
END_REGION

REGION Network 31: LD_01 - Lime vibrator / LD01
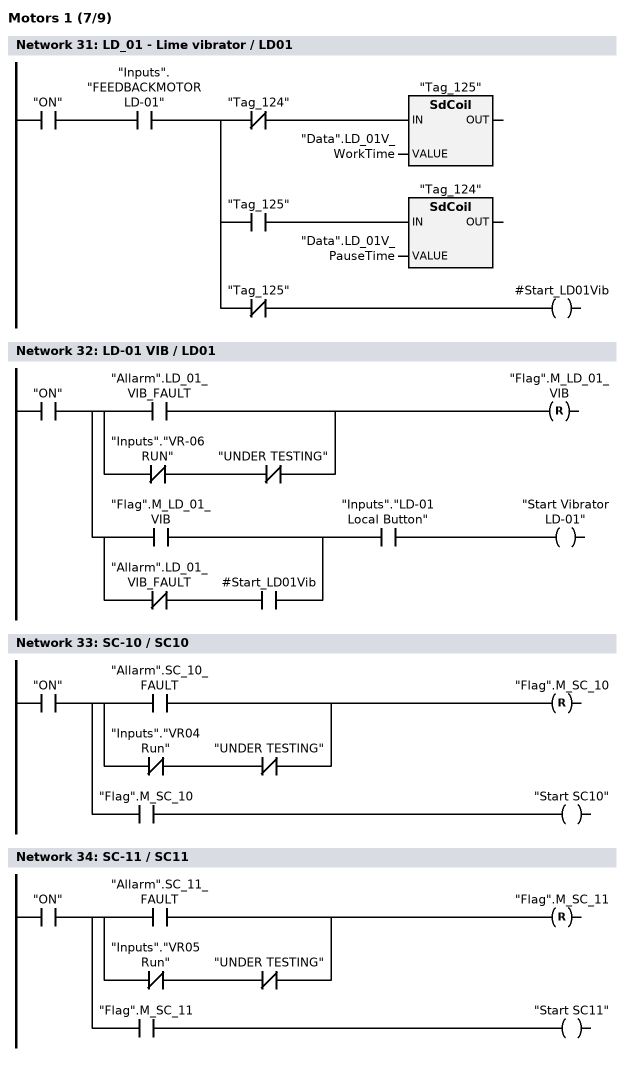
   // no SCL statement known for SdCoil: written as a call
   #_w1 := "ON" AND "Inputs"."FEEDBACKMOTOR LD-01";
   SdCoil(in := #_w1 AND NOT "Tag_124", value := "Data".LD_01V_WorkTime, operand := "Tag_125");
   SdCoil(in := #_w1 AND "Tag_125", value := "Data".LD_01V_PauseTime, operand := "Tag_124");
   #Start_LD01Vib := #_w1 AND NOT "Tag_125";
END_REGION

REGION Network 32: LD-01 VIB / LD01
   RUNG wire#powerrail
      Contact( "ON" )
      wire#w1
      Contact( "Allarm".LD_01_VIB_FAULT )
      wire#w2
      R_Coil( "Flag".M_LD_01_VIB )
   END_RUNG
   RUNG wire#w1
      I_Contact( "Inputs"."VR-06 RUN" )
      I_Contact( "UNDER TESTING" )
   END_RUNG wire#w2
   RUNG wire#w1
      Contact( "Flag".M_LD_01_VIB )
      wire#w3
      Contact( "Inputs"."LD-01 Local Button" )
      Coil( "Start Vibrator LD-01" )
   END_RUNG
   RUNG wire#w1
      I_Contact( "Allarm".LD_01_VIB_FAULT )
      Contact( #Start_LD01Vib )
   END_RUNG wire#w3
   // the same network as SCL:
   IF "ON" AND ("Allarm".LD_01_VIB_FAULT OR (NOT "Inputs"."VR-06 RUN" AND NOT "UNDER TESTING")) THEN
       "Flag".M_LD_01_VIB := FALSE;
   END_IF;
   "Start Vibrator LD-01" := "ON" AND ("Flag".M_LD_01_VIB OR (NOT "Allarm".LD_01_VIB_FAULT AND #Start_LD01Vib)) AND "Inputs"."LD-01 Local Button";
END_REGION

REGION Network 33: SC-10 / SC10
   RUNG wire#powerrail
      Contact( "ON" )
      wire#w1
      Contact( "Allarm".SC_10_FAULT )
      wire#w2
      R_Coil( "Flag".M_SC_10 )
   END_RUNG
   RUNG wire#w1
      I_Contact( "Inputs"."VR04 Run" )
      I_Contact( "UNDER TESTING" )
   END_RUNG wire#w2
   RUNG wire#w1
      Contact( "Flag".M_SC_10 )
      Coil( "Start SC10" )
   END_RUNG
   // the same network as SCL:
   IF "ON" AND ("Allarm".SC_10_FAULT OR (NOT "Inputs"."VR04 Run" AND NOT "UNDER TESTING")) THEN
       "Flag".M_SC_10 := FALSE;
   END_IF;
   "Start SC10" := "ON" AND "Flag".M_SC_10;
END_REGION

REGION Network 34: SC-11 / SC11
   RUNG wire#powerrail
      Contact( "ON" )
      wire#w1
      Contact( "Allarm".SC_11_FAULT )
      wire#w2
      R_Coil( "Flag".M_SC_11 )
   END_RUNG
   RUNG wire#w1
      I_Contact( "Inputs"."VR05 Run" )
      I_Contact( "UNDER TESTING" )
   END_RUNG wire#w2
   RUNG wire#w1
      Contact( "Flag".M_SC_11 )
      Coil( "Start SC11" )
   END_RUNG
   // the same network as SCL:
   IF "ON" AND ("Allarm".SC_11_FAULT OR (NOT "Inputs"."VR05 Run" AND NOT "UNDER TESTING")) THEN
       "Flag".M_SC_11 := FALSE;
   END_IF;
   "Start SC11" := "ON" AND "Flag".M_SC_11;
END_REGION

REGION Network 35: Stop FN-04 if alarms persistance / PREALLARM FN04
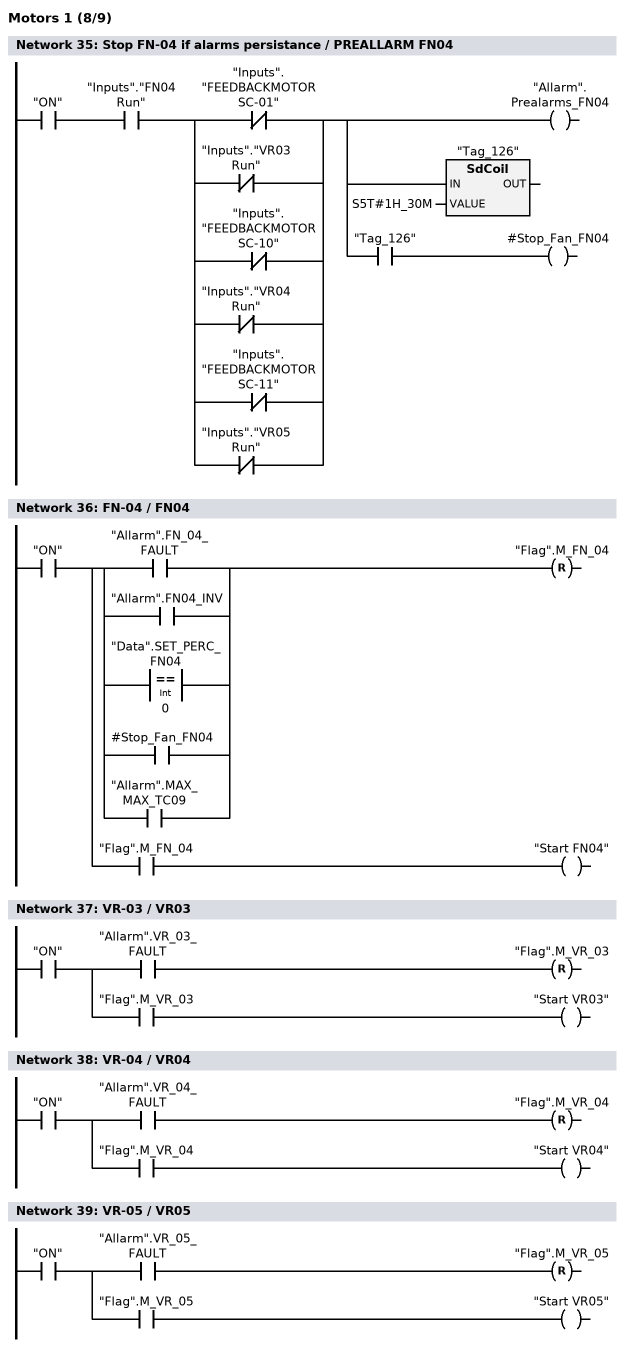
   // no SCL statement known for SdCoil: written as a call
   "Allarm".Prealarms_FN04 := "ON" AND "Inputs"."FN04 Run" AND (NOT "Inputs"."FEEDBACKMOTOR SC-01" OR NOT "Inputs"."VR03 Run" OR NOT "Inputs"."FEEDBACKMOTOR SC-10" OR NOT "Inputs"."VR04 Run" OR NOT "Inputs"."FEEDBACKMOTOR SC-11" OR NOT "Inputs"."VR05 Run");
   #_w1 := "Allarm".Prealarms_FN04;
   SdCoil(in := "Allarm".Prealarms_FN04, value := S5T#1H_30M, operand := "Tag_126");
   #Stop_Fan_FN04 := #_w1 AND "Tag_126";
END_REGION

REGION Network 36: FN-04 / FN04
   RUNG wire#powerrail
      Contact( "ON" )
      wire#w1
      Contact( "Allarm".FN_04_FAULT )
      wire#w2
      R_Coil( "Flag".M_FN_04 )
   END_RUNG
   RUNG wire#w1
      Contact( "Allarm".FN04_INV )
   END_RUNG wire#w2
   RUNG wire#w1
      { S7_Templates := "SrcType := Int" } EQ_Contact(in1 := "Data".SET_PERC_FN04, in2 := 0)
   END_RUNG wire#w2
   RUNG wire#w1
      Contact( #Stop_Fan_FN04 )
   END_RUNG wire#w2
   RUNG wire#w1
      Contact( "Allarm".MAX_MAX_TC09 )
   END_RUNG wire#w2
   RUNG wire#w1
      Contact( "Flag".M_FN_04 )
      Coil( "Start FN04" )
   END_RUNG
   // the same network as SCL:
   IF "ON" AND ("Allarm".FN_04_FAULT OR "Allarm".FN04_INV OR ("Data".SET_PERC_FN04 = 0) OR #Stop_Fan_FN04 OR "Allarm".MAX_MAX_TC09) THEN
       "Flag".M_FN_04 := FALSE;
   END_IF;
   "Start FN04" := "ON" AND "Flag".M_FN_04;
END_REGION

REGION Network 37: VR-03 / VR03
   RUNG wire#powerrail
      Contact( "ON" )
      wire#w1
      Contact( "Allarm".VR_03_FAULT )
      R_Coil( "Flag".M_VR_03 )
   END_RUNG
   RUNG wire#w1
      Contact( "Flag".M_VR_03 )
      Coil( "Start VR03" )
   END_RUNG
   // the same network as SCL:
   IF "ON" AND "Allarm".VR_03_FAULT THEN "Flag".M_VR_03 := FALSE; END_IF;
   "Start VR03" := "ON" AND "Flag".M_VR_03;
END_REGION

REGION Network 38: VR-04 / VR04
   RUNG wire#powerrail
      Contact( "ON" )
      wire#w1
      Contact( "Allarm".VR_04_FAULT )
      R_Coil( "Flag".M_VR_04 )
   END_RUNG
   RUNG wire#w1
      Contact( "Flag".M_VR_04 )
      Coil( "Start VR04" )
   END_RUNG
   // the same network as SCL:
   IF "ON" AND "Allarm".VR_04_FAULT THEN "Flag".M_VR_04 := FALSE; END_IF;
   "Start VR04" := "ON" AND "Flag".M_VR_04;
END_REGION

REGION Network 39: VR-05 / VR05
   RUNG wire#powerrail
      Contact( "ON" )
      wire#w1
      Contact( "Allarm".VR_05_FAULT )
      R_Coil( "Flag".M_VR_05 )
   END_RUNG
   RUNG wire#w1
      Contact( "Flag".M_VR_05 )
      Coil( "Start VR05" )
   END_RUNG
   // the same network as SCL:
   IF "ON" AND "Allarm".VR_05_FAULT THEN "Flag".M_VR_05 := FALSE; END_IF;
   "Start VR05" := "ON" AND "Flag".M_VR_05;
END_REGION

REGION Network 40: VR-06 / VR06
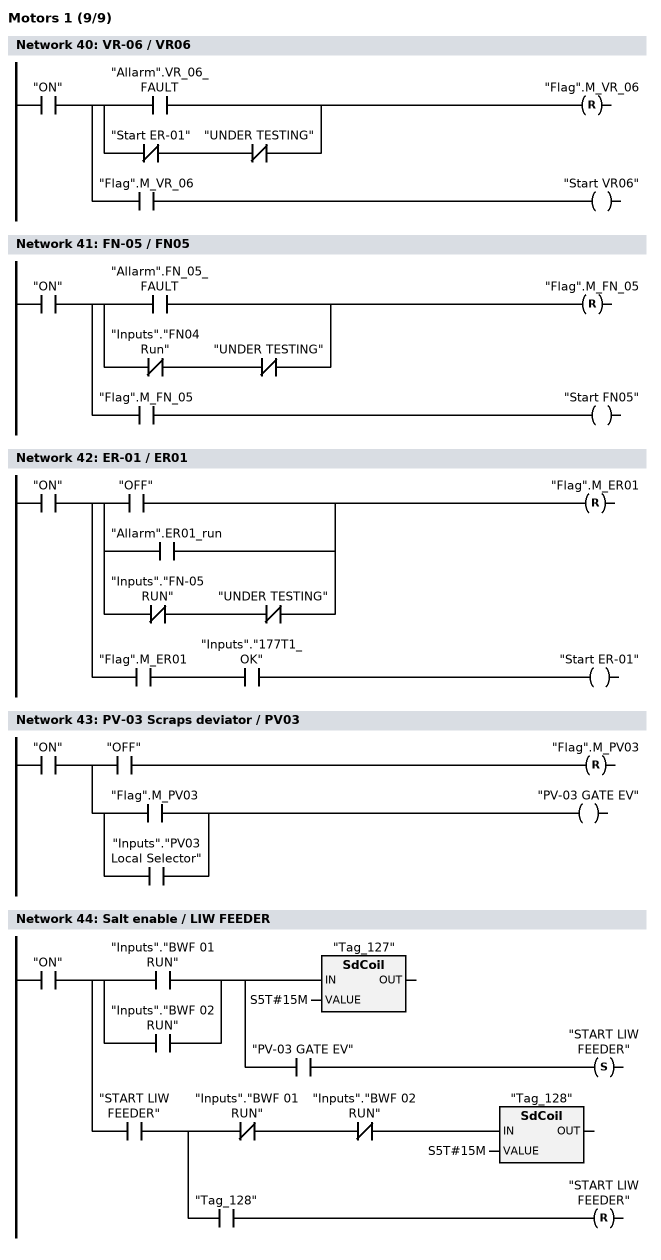
   RUNG wire#powerrail
      Contact( "ON" )
      wire#w1
      Contact( "Allarm".VR_06_FAULT )
      wire#w2
      R_Coil( "Flag".M_VR_06 )
   END_RUNG
   RUNG wire#w1
      I_Contact( "Start ER-01" )
      I_Contact( "UNDER TESTING" )
   END_RUNG wire#w2
   RUNG wire#w1
      Contact( "Flag".M_VR_06 )
      Coil( "Start VR06" )
   END_RUNG
   // the same network as SCL:
   IF "ON" AND ("Allarm".VR_06_FAULT OR (NOT "Start ER-01" AND NOT "UNDER TESTING")) THEN
       "Flag".M_VR_06 := FALSE;
   END_IF;
   "Start VR06" := "ON" AND "Flag".M_VR_06;
END_REGION

REGION Network 41: FN-05 / FN05
   RUNG wire#powerrail
      Contact( "ON" )
      wire#w1
      Contact( "Allarm".FN_05_FAULT )
      wire#w2
      R_Coil( "Flag".M_FN_05 )
   END_RUNG
   RUNG wire#w1
      I_Contact( "Inputs"."FN04 Run" )
      I_Contact( "UNDER TESTING" )
   END_RUNG wire#w2
   RUNG wire#w1
      Contact( "Flag".M_FN_05 )
      Coil( "Start FN05" )
   END_RUNG
   // the same network as SCL:
   IF "ON" AND ("Allarm".FN_05_FAULT OR (NOT "Inputs"."FN04 Run" AND NOT "UNDER TESTING")) THEN
       "Flag".M_FN_05 := FALSE;
   END_IF;
   "Start FN05" := "ON" AND "Flag".M_FN_05;
END_REGION

REGION Network 42: ER-01 / ER01
   RUNG wire#powerrail
      Contact( "ON" )
      wire#w1
      Contact( "OFF" )
      wire#w2
      R_Coil( "Flag".M_ER01 )
   END_RUNG
   RUNG wire#w1
      Contact( "Allarm".ER01_run )
   END_RUNG wire#w2
   RUNG wire#w1
      I_Contact( "Inputs"."FN-05 RUN" )
      I_Contact( "UNDER TESTING" )
   END_RUNG wire#w2
   RUNG wire#w1
      Contact( "Flag".M_ER01 )
      Contact( "Inputs"."177T1_OK" )
      Coil( "Start ER-01" )
   END_RUNG
   // the same network as SCL:
   IF "ON" AND ("OFF" OR "Allarm".ER01_run OR (NOT "Inputs"."FN-05 RUN" AND NOT "UNDER TESTING")) THEN
       "Flag".M_ER01 := FALSE;
   END_IF;
   "Start ER-01" := "ON" AND "Flag".M_ER01 AND "Inputs"."177T1_OK";
END_REGION

REGION Network 43: PV-03 Scraps deviator / PV03
   RUNG wire#powerrail
      Contact( "ON" )
      wire#w1
      Contact( "OFF" )
      R_Coil( "Flag".M_PV03 )
   END_RUNG
   RUNG wire#w1
      Contact( "Flag".M_PV03 )
      wire#w2
      Coil( "PV-03 GATE EV" )
   END_RUNG
   RUNG wire#w1
      Contact( "Inputs"."PV03 Local Selector" )
   END_RUNG wire#w2
   // the same network as SCL:
   IF "ON" AND "OFF" THEN "Flag".M_PV03 := FALSE; END_IF;
   "PV-03 GATE EV" := "ON" AND ("Flag".M_PV03 OR "Inputs"."PV03 Local Selector");
END_REGION

REGION Network 44: Salt enable / LIW FEEDER
   // no SCL statement known for SdCoil: written as a call
   #_w1 := "ON" AND ("Inputs"."BWF 01 RUN" OR "Inputs"."BWF 02 RUN");
   #_w2 := "ON";
   SdCoil(in := #_w1, value := S5T#15M, operand := "Tag_127");
   IF #_w1 AND "PV-03 GATE EV" THEN "START LIW FEEDER" := TRUE; END_IF;
   #_w3 := #_w2 AND "START LIW FEEDER";
   SdCoil(in := #_w3 AND NOT "Inputs"."BWF 01 RUN" AND NOT "Inputs"."BWF 02 RUN",
          value := S5T#15M,
          operand := "Tag_128");
   IF #_w3 AND "Tag_128" THEN "START LIW FEEDER" := FALSE; END_IF;
END_REGION
END_FUNCTION

FUNCTION "Filter" : Void   // FC8, LAD
TITLE = Gestione battute filtri / Management of filter beats
{ S7_Optimized_Access := 'FALSE' }
VERSION : 0.1
   VAR_TEMP
      app01 : Int;
      App02 : Int;
      Abilita_lavaggio_BF01 : Bool;
      Abilita_lavaggio_BF02 : Bool;
      Forza_Lavaggio : Bool;
      App_Word : Word;
   END_VAR
   VAR_TEMP   // added for the SCL form of the ladder/FBD networks
      _w1 : Bool;
      _w2 : Bool;
   END_VAR
BEGIN

REGION Network 1
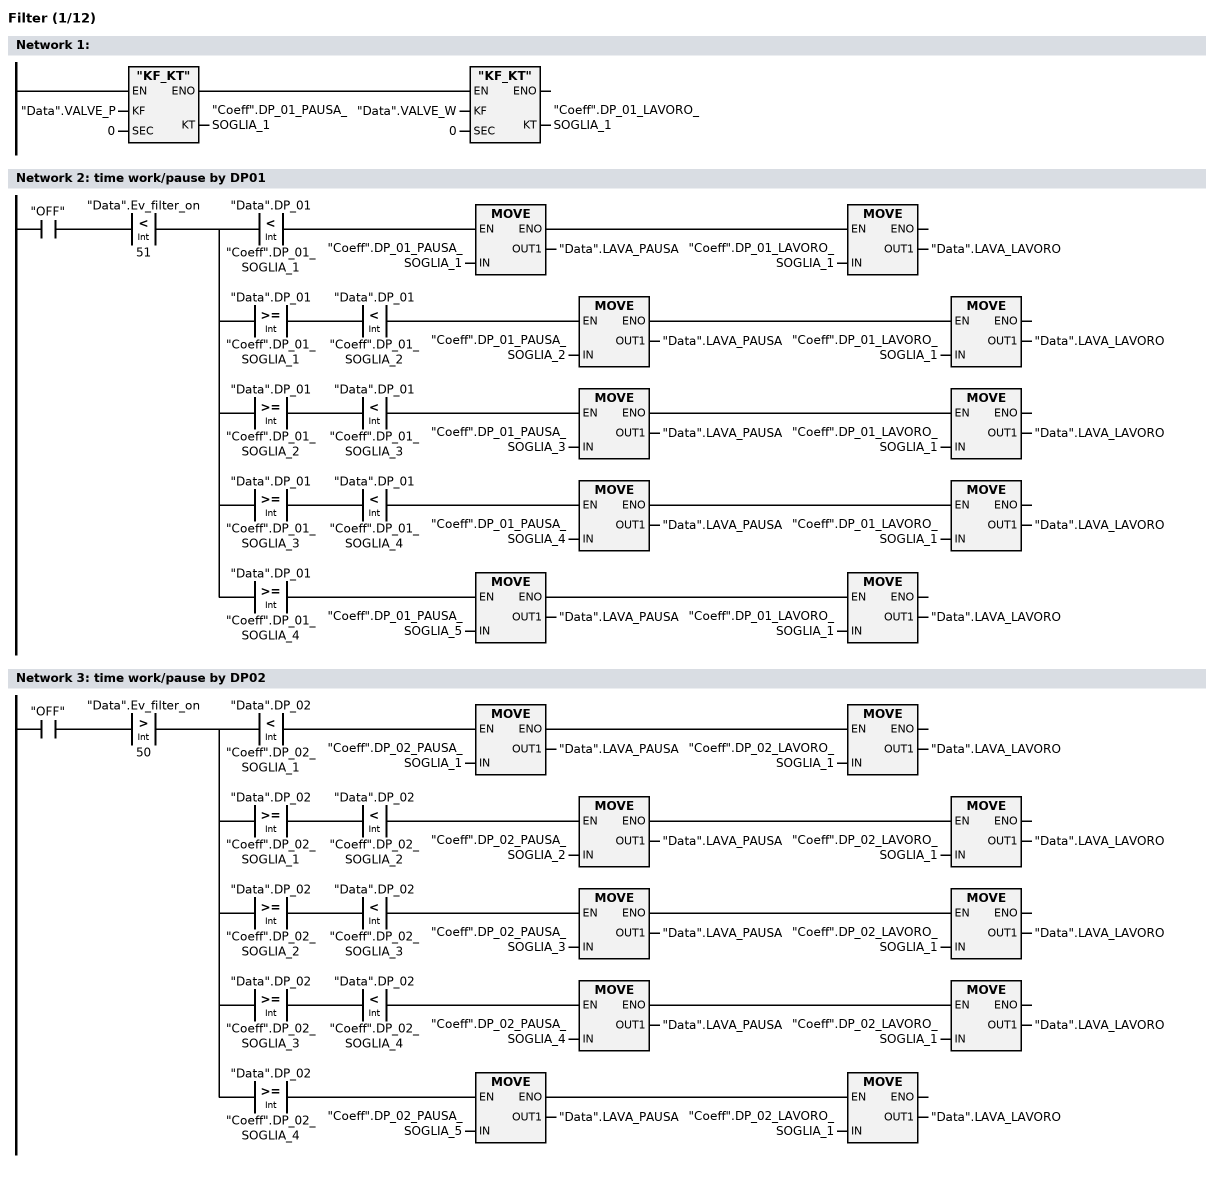
   RUNG wire#powerrail
      "KF_KT"(KF := "Data".VALVE_P, SEC := 0, KT => "Coeff".DP_01_PAUSA_SOGLIA_1)
      "KF_KT"(KF := "Data".VALVE_W, SEC := 0, KT => "Coeff".DP_01_LAVORO_SOGLIA_1)
   END_RUNG
   // the same network as SCL:
   "KF_KT"(KF := "Data".VALVE_P, SEC := 0, KT => "Coeff".DP_01_PAUSA_SOGLIA_1, ENO => #_w1);
   IF #_w1 THEN "KF_KT"(KF := "Data".VALVE_W, SEC := 0, KT => "Coeff".DP_01_LAVORO_SOGLIA_1); END_IF;
END_REGION

REGION Network 2: time work/pause by DP01
   RUNG wire#powerrail
      Contact( "OFF" )
      { S7_Templates := "SrcType := Int" } LT_Contact(in1 := "Data".Ev_filter_on, in2 := 51)
      wire#w1
      { S7_Templates := "SrcType := Int" } LT_Contact(in1 := "Data".DP_01, in2 := "Coeff".DP_01_SOGLIA_1)
      { S7_GenerateENO := "TRUE" } Move(in := "Coeff".DP_01_PAUSA_SOGLIA_1, out1 => "Data".LAVA_PAUSA)
      { S7_GenerateENO := "TRUE" } Move(in := "Coeff".DP_01_LAVORO_SOGLIA_1, out1 => "Data".LAVA_LAVORO)
   END_RUNG
   RUNG wire#w1
      { S7_Templates := "SrcType := Int" } GE_Contact(in1 := "Data".DP_01, in2 := "Coeff".DP_01_SOGLIA_1)
      { S7_Templates := "SrcType := Int" } LT_Contact(in1 := "Data".DP_01, in2 := "Coeff".DP_01_SOGLIA_2)
      { S7_GenerateENO := "TRUE" } Move(in := "Coeff".DP_01_PAUSA_SOGLIA_2, out1 => "Data".LAVA_PAUSA)
      { S7_GenerateENO := "TRUE" } Move(in := "Coeff".DP_01_LAVORO_SOGLIA_1, out1 => "Data".LAVA_LAVORO)
   END_RUNG
   RUNG wire#w1
      { S7_Templates := "SrcType := Int" } GE_Contact(in1 := "Data".DP_01, in2 := "Coeff".DP_01_SOGLIA_2)
      { S7_Templates := "SrcType := Int" } LT_Contact(in1 := "Data".DP_01, in2 := "Coeff".DP_01_SOGLIA_3)
      { S7_GenerateENO := "TRUE" } Move(in := "Coeff".DP_01_PAUSA_SOGLIA_3, out1 => "Data".LAVA_PAUSA)
      { S7_GenerateENO := "TRUE" } Move(in := "Coeff".DP_01_LAVORO_SOGLIA_1, out1 => "Data".LAVA_LAVORO)
   END_RUNG
   RUNG wire#w1
      { S7_Templates := "SrcType := Int" } GE_Contact(in1 := "Data".DP_01, in2 := "Coeff".DP_01_SOGLIA_3)
      { S7_Templates := "SrcType := Int" } LT_Contact(in1 := "Data".DP_01, in2 := "Coeff".DP_01_SOGLIA_4)
      { S7_GenerateENO := "TRUE" } Move(in := "Coeff".DP_01_PAUSA_SOGLIA_4, out1 => "Data".LAVA_PAUSA)
      { S7_GenerateENO := "TRUE" } Move(in := "Coeff".DP_01_LAVORO_SOGLIA_1, out1 => "Data".LAVA_LAVORO)
   END_RUNG
   RUNG wire#w1
      { S7_Templates := "SrcType := Int" } GE_Contact(in1 := "Data".DP_01, in2 := "Coeff".DP_01_SOGLIA_4)
      { S7_GenerateENO := "TRUE" } Move(in := "Coeff".DP_01_PAUSA_SOGLIA_5, out1 => "Data".LAVA_PAUSA)
      { S7_GenerateENO := "TRUE" } Move(in := "Coeff".DP_01_LAVORO_SOGLIA_1, out1 => "Data".LAVA_LAVORO)
   END_RUNG
   // the same network as SCL:
   // ENO of a box is taken as its EN; it also drops when the box reports an error
   #_w1 := "OFF" AND ("Data".Ev_filter_on < 51);
   IF #_w1 AND ("Data".DP_01 < "Coeff".DP_01_SOGLIA_1) THEN
       "Data".LAVA_PAUSA := "Coeff".DP_01_PAUSA_SOGLIA_1;
       "Data".LAVA_LAVORO := "Coeff".DP_01_LAVORO_SOGLIA_1;
   END_IF;
   IF #_w1 AND ("Data".DP_01 >= "Coeff".DP_01_SOGLIA_1) AND ("Data".DP_01 < "Coeff".DP_01_SOGLIA_2) THEN
       "Data".LAVA_PAUSA := "Coeff".DP_01_PAUSA_SOGLIA_2;
       "Data".LAVA_LAVORO := "Coeff".DP_01_LAVORO_SOGLIA_1;
   END_IF;
   IF #_w1 AND ("Data".DP_01 >= "Coeff".DP_01_SOGLIA_2) AND ("Data".DP_01 < "Coeff".DP_01_SOGLIA_3) THEN
       "Data".LAVA_PAUSA := "Coeff".DP_01_PAUSA_SOGLIA_3;
       "Data".LAVA_LAVORO := "Coeff".DP_01_LAVORO_SOGLIA_1;
   END_IF;
   IF #_w1 AND ("Data".DP_01 >= "Coeff".DP_01_SOGLIA_3) AND ("Data".DP_01 < "Coeff".DP_01_SOGLIA_4) THEN
       "Data".LAVA_PAUSA := "Coeff".DP_01_PAUSA_SOGLIA_4;
       "Data".LAVA_LAVORO := "Coeff".DP_01_LAVORO_SOGLIA_1;
   END_IF;
   IF #_w1 AND ("Data".DP_01 >= "Coeff".DP_01_SOGLIA_4) THEN
       "Data".LAVA_PAUSA := "Coeff".DP_01_PAUSA_SOGLIA_5;
       "Data".LAVA_LAVORO := "Coeff".DP_01_LAVORO_SOGLIA_1;
   END_IF;
END_REGION

REGION Network 3: time work/pause by DP02
   RUNG wire#powerrail
      Contact( "OFF" )
      { S7_Templates := "SrcType := Int" } GT_Contact(in1 := "Data".Ev_filter_on, in2 := 50)
      wire#w1
      { S7_Templates := "SrcType := Int" } LT_Contact(in1 := "Data".DP_02, in2 := "Coeff".DP_02_SOGLIA_1)
      { S7_GenerateENO := "TRUE" } Move(in := "Coeff".DP_02_PAUSA_SOGLIA_1, out1 => "Data".LAVA_PAUSA)
      { S7_GenerateENO := "TRUE" } Move(in := "Coeff".DP_02_LAVORO_SOGLIA_1, out1 => "Data".LAVA_LAVORO)
   END_RUNG
   RUNG wire#w1
      { S7_Templates := "SrcType := Int" } GE_Contact(in1 := "Data".DP_02, in2 := "Coeff".DP_02_SOGLIA_1)
      { S7_Templates := "SrcType := Int" } LT_Contact(in1 := "Data".DP_02, in2 := "Coeff".DP_02_SOGLIA_2)
      { S7_GenerateENO := "TRUE" } Move(in := "Coeff".DP_02_PAUSA_SOGLIA_2, out1 => "Data".LAVA_PAUSA)
      { S7_GenerateENO := "TRUE" } Move(in := "Coeff".DP_02_LAVORO_SOGLIA_1, out1 => "Data".LAVA_LAVORO)
   END_RUNG
   RUNG wire#w1
      { S7_Templates := "SrcType := Int" } GE_Contact(in1 := "Data".DP_02, in2 := "Coeff".DP_02_SOGLIA_2)
      { S7_Templates := "SrcType := Int" } LT_Contact(in1 := "Data".DP_02, in2 := "Coeff".DP_02_SOGLIA_3)
      { S7_GenerateENO := "TRUE" } Move(in := "Coeff".DP_02_PAUSA_SOGLIA_3, out1 => "Data".LAVA_PAUSA)
      { S7_GenerateENO := "TRUE" } Move(in := "Coeff".DP_02_LAVORO_SOGLIA_1, out1 => "Data".LAVA_LAVORO)
   END_RUNG
   RUNG wire#w1
      { S7_Templates := "SrcType := Int" } GE_Contact(in1 := "Data".DP_02, in2 := "Coeff".DP_02_SOGLIA_3)
      { S7_Templates := "SrcType := Int" } LT_Contact(in1 := "Data".DP_02, in2 := "Coeff".DP_02_SOGLIA_4)
      { S7_GenerateENO := "TRUE" } Move(in := "Coeff".DP_02_PAUSA_SOGLIA_4, out1 => "Data".LAVA_PAUSA)
      { S7_GenerateENO := "TRUE" } Move(in := "Coeff".DP_02_LAVORO_SOGLIA_1, out1 => "Data".LAVA_LAVORO)
   END_RUNG
   RUNG wire#w1
      { S7_Templates := "SrcType := Int" } GE_Contact(in1 := "Data".DP_02, in2 := "Coeff".DP_02_SOGLIA_4)
      { S7_GenerateENO := "TRUE" } Move(in := "Coeff".DP_02_PAUSA_SOGLIA_5, out1 => "Data".LAVA_PAUSA)
      { S7_GenerateENO := "TRUE" } Move(in := "Coeff".DP_02_LAVORO_SOGLIA_1, out1 => "Data".LAVA_LAVORO)
   END_RUNG
   // the same network as SCL:
   // ENO of a box is taken as its EN; it also drops when the box reports an error
   #_w1 := "OFF" AND ("Data".Ev_filter_on > 50);
   IF #_w1 AND ("Data".DP_02 < "Coeff".DP_02_SOGLIA_1) THEN
       "Data".LAVA_PAUSA := "Coeff".DP_02_PAUSA_SOGLIA_1;
       "Data".LAVA_LAVORO := "Coeff".DP_02_LAVORO_SOGLIA_1;
   END_IF;
   IF #_w1 AND ("Data".DP_02 >= "Coeff".DP_02_SOGLIA_1) AND ("Data".DP_02 < "Coeff".DP_02_SOGLIA_2) THEN
       "Data".LAVA_PAUSA := "Coeff".DP_02_PAUSA_SOGLIA_2;
       "Data".LAVA_LAVORO := "Coeff".DP_02_LAVORO_SOGLIA_1;
   END_IF;
   IF #_w1 AND ("Data".DP_02 >= "Coeff".DP_02_SOGLIA_2) AND ("Data".DP_02 < "Coeff".DP_02_SOGLIA_3) THEN
       "Data".LAVA_PAUSA := "Coeff".DP_02_PAUSA_SOGLIA_3;
       "Data".LAVA_LAVORO := "Coeff".DP_02_LAVORO_SOGLIA_1;
   END_IF;
   IF #_w1 AND ("Data".DP_02 >= "Coeff".DP_02_SOGLIA_3) AND ("Data".DP_02 < "Coeff".DP_02_SOGLIA_4) THEN
       "Data".LAVA_PAUSA := "Coeff".DP_02_PAUSA_SOGLIA_4;
       "Data".LAVA_LAVORO := "Coeff".DP_02_LAVORO_SOGLIA_1;
   END_IF;
   IF #_w1 AND ("Data".DP_02 >= "Coeff".DP_02_SOGLIA_4) THEN
       "Data".LAVA_PAUSA := "Coeff".DP_02_PAUSA_SOGLIA_5;
       "Data".LAVA_LAVORO := "Coeff".DP_02_LAVORO_SOGLIA_1;
   END_IF;
END_REGION

REGION Network 4: Forza lavaggio minimo / Force wash minimum
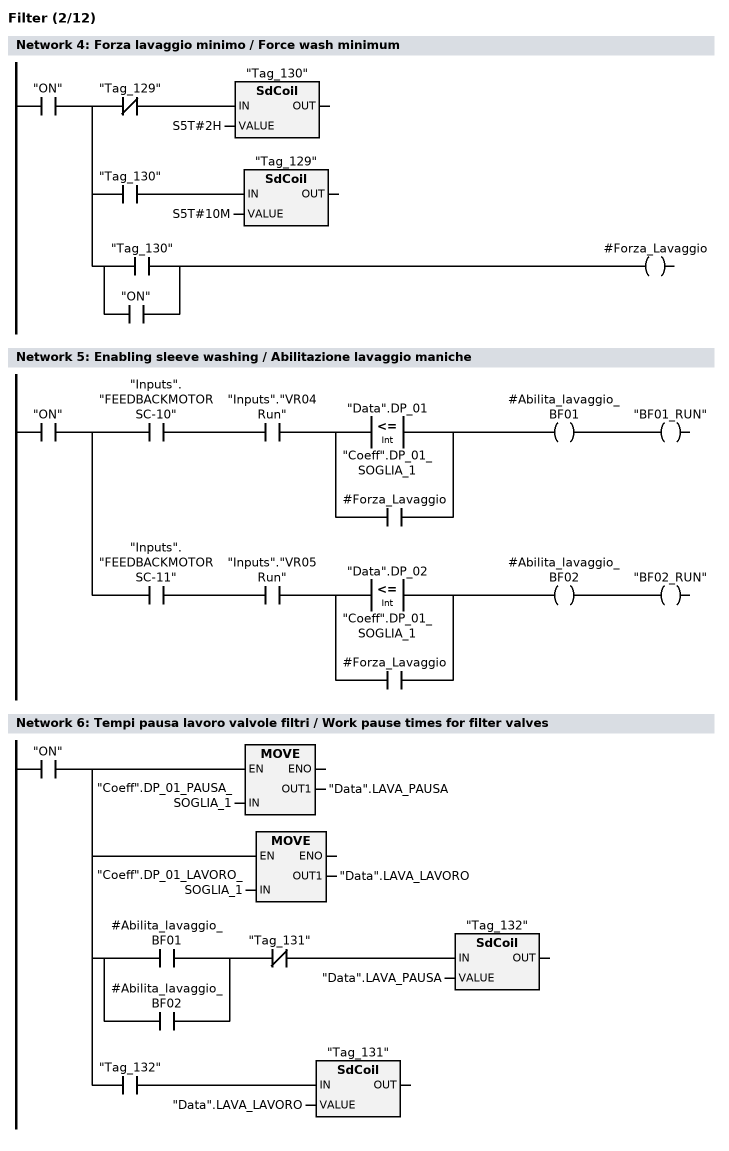
   // no SCL statement known for SdCoil: written as a call
   #_w1 := "ON";
   SdCoil(in := "ON" AND NOT "Tag_129", value := S5T#2H, operand := "Tag_130");
   SdCoil(in := #_w1 AND "Tag_130", value := S5T#10M, operand := "Tag_129");
   #Forza_Lavaggio := #_w1 AND ("Tag_130" OR "ON");
END_REGION

REGION Network 5: Enabling sleeve washing / Abilitazione lavaggio maniche
   RUNG wire#powerrail
      Contact( "ON" )
      wire#w1
      Contact( "Inputs"."FEEDBACKMOTOR SC-10" )
      Contact( "Inputs"."VR04 Run" )
      wire#w2
      { S7_Templates := "SrcType := Int" } LE_Contact(in1 := "Data".DP_01, in2 := "Coeff".DP_01_SOGLIA_1)
      wire#w3
      Coil( #Abilita_lavaggio_BF01 )
      Coil( "BF01_RUN" )
   END_RUNG
   RUNG wire#w2
      Contact( #Forza_Lavaggio )
   END_RUNG wire#w3
   RUNG wire#w1
      Contact( "Inputs"."FEEDBACKMOTOR SC-11" )
      Contact( "Inputs"."VR05 Run" )
      wire#w4
      { S7_Templates := "SrcType := Int" } LE_Contact(in1 := "Data".DP_02, in2 := "Coeff".DP_01_SOGLIA_1)
      wire#w5
      Coil( #Abilita_lavaggio_BF02 )
      Coil( "BF02_RUN" )
   END_RUNG
   RUNG wire#w4
      Contact( #Forza_Lavaggio )
   END_RUNG wire#w5
   // the same network as SCL:
   #Abilita_lavaggio_BF01 := "ON" AND "Inputs"."FEEDBACKMOTOR SC-10" AND "Inputs"."VR04 Run" AND (("Data".DP_01 <= "Coeff".DP_01_SOGLIA_1) OR #Forza_Lavaggio);
   "BF01_RUN" := #Abilita_lavaggio_BF01;
   #Abilita_lavaggio_BF02 := "ON" AND "Inputs"."FEEDBACKMOTOR SC-11" AND "Inputs"."VR05 Run" AND (("Data".DP_02 <= "Coeff".DP_01_SOGLIA_1) OR #Forza_Lavaggio);
   "BF02_RUN" := #Abilita_lavaggio_BF02;
END_REGION

REGION Network 6: Tempi pausa lavoro valvole filtri / Work pause times for filter valves
   // no SCL statement known for SdCoil: written as a call
   IF "ON" THEN
       "Data".LAVA_PAUSA := "Coeff".DP_01_PAUSA_SOGLIA_1;
       "Data".LAVA_LAVORO := "Coeff".DP_01_LAVORO_SOGLIA_1;
   END_IF;
   #_w1 := "ON";
   SdCoil(in := "ON" AND (#Abilita_lavaggio_BF01 OR #Abilita_lavaggio_BF02) AND NOT "Tag_131",
          value := "Data".LAVA_PAUSA,
          operand := "Tag_132");
   SdCoil(in := #_w1 AND "Tag_132", value := "Data".LAVA_LAVORO, operand := "Tag_131");
END_REGION

REGION Network 7: filter work
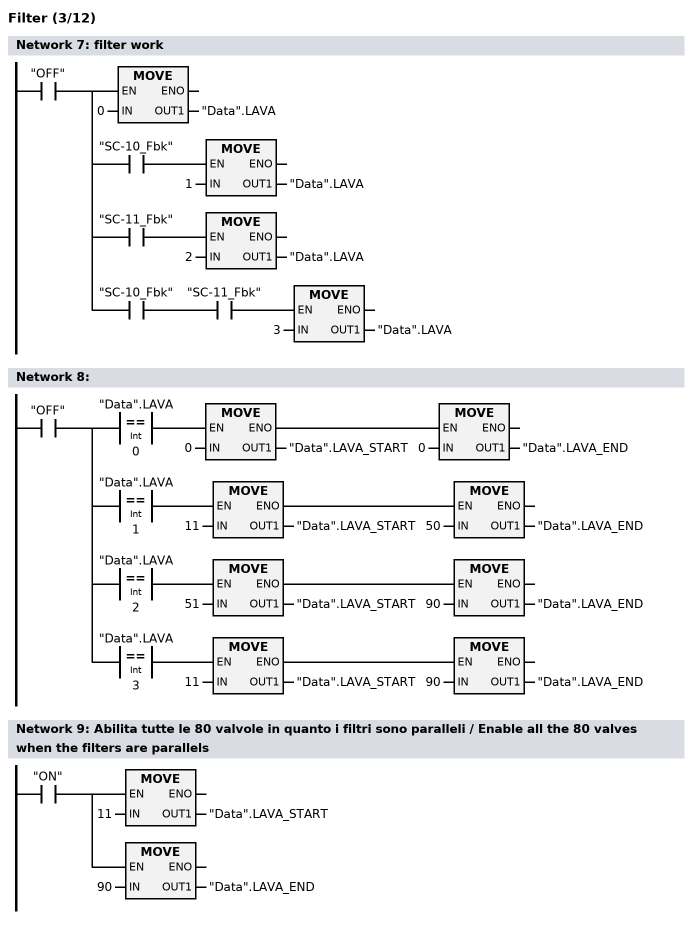
   RUNG wire#powerrail
      Contact( "OFF" )
      wire#w1
      { S7_GenerateENO := "TRUE" } Move(in := 0, out1 => "Data".LAVA)
   END_RUNG
   RUNG wire#w1
      Contact( "SC-10_Fbk" )
      { S7_GenerateENO := "TRUE" } Move(in := 1, out1 => "Data".LAVA)
   END_RUNG
   RUNG wire#w1
      Contact( "SC-11_Fbk" )
      { S7_GenerateENO := "TRUE" } Move(in := 2, out1 => "Data".LAVA)
   END_RUNG
   RUNG wire#w1
      Contact( "SC-10_Fbk" )
      Contact( "SC-11_Fbk" )
      { S7_GenerateENO := "TRUE" } Move(in := 3, out1 => "Data".LAVA)
   END_RUNG
   // the same network as SCL:
   IF "OFF" THEN "Data".LAVA := 0; END_IF;
   IF "OFF" AND "SC-10_Fbk" THEN "Data".LAVA := 1; END_IF;
   IF "OFF" AND "SC-11_Fbk" THEN "Data".LAVA := 2; END_IF;
   IF "OFF" AND "SC-10_Fbk" AND "SC-11_Fbk" THEN "Data".LAVA := 3; END_IF;
END_REGION

REGION Network 8
   RUNG wire#powerrail
      Contact( "OFF" )
      wire#w1
      { S7_Templates := "SrcType := Int" } EQ_Contact(in1 := "Data".LAVA, in2 := 0)
      { S7_GenerateENO := "TRUE" } Move(in := 0, out1 => "Data".LAVA_START)
      { S7_GenerateENO := "TRUE" } Move(in := 0, out1 => "Data".LAVA_END)
   END_RUNG
   RUNG wire#w1
      { S7_Templates := "SrcType := Int" } EQ_Contact(in1 := "Data".LAVA, in2 := 1)
      { S7_GenerateENO := "TRUE" } Move(in := 11, out1 => "Data".LAVA_START)
      { S7_GenerateENO := "TRUE" } Move(in := 50, out1 => "Data".LAVA_END)
   END_RUNG
   RUNG wire#w1
      { S7_Templates := "SrcType := Int" } EQ_Contact(in1 := "Data".LAVA, in2 := 2)
      { S7_GenerateENO := "TRUE" } Move(in := 51, out1 => "Data".LAVA_START)
      { S7_GenerateENO := "TRUE" } Move(in := 90, out1 => "Data".LAVA_END)
   END_RUNG
   RUNG wire#w1
      { S7_Templates := "SrcType := Int" } EQ_Contact(in1 := "Data".LAVA, in2 := 3)
      { S7_GenerateENO := "TRUE" } Move(in := 11, out1 => "Data".LAVA_START)
      { S7_GenerateENO := "TRUE" } Move(in := 90, out1 => "Data".LAVA_END)
   END_RUNG
   // the same network as SCL:
   // ENO of a box is taken as its EN; it also drops when the box reports an error
   IF "OFF" AND ("Data".LAVA = 0) THEN
       "Data".LAVA_START := 0;
       "Data".LAVA_END := 0;
   END_IF;
   IF "OFF" AND ("Data".LAVA = 1) THEN
       "Data".LAVA_START := 11;
       "Data".LAVA_END := 50;
   END_IF;
   IF "OFF" AND ("Data".LAVA = 2) THEN
       "Data".LAVA_START := 51;
       "Data".LAVA_END := 90;
   END_IF;
   IF "OFF" AND ("Data".LAVA = 3) THEN
       "Data".LAVA_START := 11;
       "Data".LAVA_END := 90;
   END_IF;
END_REGION

REGION Network 9: Abilita tutte le 80 valvole in quanto i filtri sono paralleli / Enable all the 80 valves when the filters are parallels
   RUNG wire#powerrail
      Contact( "ON" )
      wire#w1
      { S7_GenerateENO := "TRUE" } Move(in := 11, out1 => "Data".LAVA_START)
   END_RUNG
   RUNG wire#w1
      { S7_GenerateENO := "TRUE" } Move(in := 90, out1 => "Data".LAVA_END)
   END_RUNG
   // the same network as SCL:
   IF "ON" THEN
       "Data".LAVA_START := 11;
       "Data".LAVA_END := 90;
   END_IF;
END_REGION

REGION Network 10: wash filter / A0.0 FILTER 1 VALVE BF01FIRST SECTOR
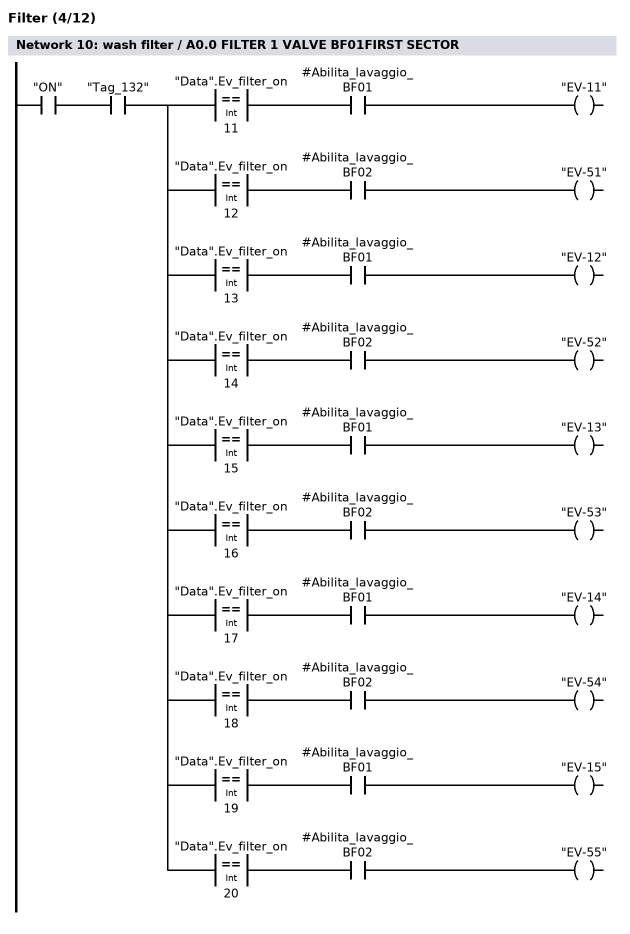
   RUNG wire#powerrail
      Contact( "ON" )
      Contact( "Tag_132" )
      wire#w1
      { S7_Templates := "SrcType := Int" } EQ_Contact(in1 := "Data".Ev_filter_on, in2 := 11)
      Contact( #Abilita_lavaggio_BF01 )
      Coil( "EV-11" )
   END_RUNG
   RUNG wire#w1
      { S7_Templates := "SrcType := Int" } EQ_Contact(in1 := "Data".Ev_filter_on, in2 := 12)
      Contact( #Abilita_lavaggio_BF02 )
      Coil( "EV-51" )
   END_RUNG
   RUNG wire#w1
      { S7_Templates := "SrcType := Int" } EQ_Contact(in1 := "Data".Ev_filter_on, in2 := 13)
      Contact( #Abilita_lavaggio_BF01 )
      Coil( "EV-12" )
   END_RUNG
   RUNG wire#w1
      { S7_Templates := "SrcType := Int" } EQ_Contact(in1 := "Data".Ev_filter_on, in2 := 14)
      Contact( #Abilita_lavaggio_BF02 )
      Coil( "EV-52" )
   END_RUNG
   RUNG wire#w1
      { S7_Templates := "SrcType := Int" } EQ_Contact(in1 := "Data".Ev_filter_on, in2 := 15)
      Contact( #Abilita_lavaggio_BF01 )
      Coil( "EV-13" )
   END_RUNG
   RUNG wire#w1
      { S7_Templates := "SrcType := Int" } EQ_Contact(in1 := "Data".Ev_filter_on, in2 := 16)
      Contact( #Abilita_lavaggio_BF02 )
      Coil( "EV-53" )
   END_RUNG
   RUNG wire#w1
      { S7_Templates := "SrcType := Int" } EQ_Contact(in1 := "Data".Ev_filter_on, in2 := 17)
      Contact( #Abilita_lavaggio_BF01 )
      Coil( "EV-14" )
   END_RUNG
   RUNG wire#w1
      { S7_Templates := "SrcType := Int" } EQ_Contact(in1 := "Data".Ev_filter_on, in2 := 18)
      Contact( #Abilita_lavaggio_BF02 )
      Coil( "EV-54" )
   END_RUNG
   RUNG wire#w1
      { S7_Templates := "SrcType := Int" } EQ_Contact(in1 := "Data".Ev_filter_on, in2 := 19)
      Contact( #Abilita_lavaggio_BF01 )
      Coil( "EV-15" )
   END_RUNG
   RUNG wire#w1
      { S7_Templates := "SrcType := Int" } EQ_Contact(in1 := "Data".Ev_filter_on, in2 := 20)
      Contact( #Abilita_lavaggio_BF02 )
      Coil( "EV-55" )
   END_RUNG
   // the same network as SCL:
   #_w1 := "ON" AND "Tag_132";
   "EV-11" := #_w1 AND ("Data".Ev_filter_on = 11) AND #Abilita_lavaggio_BF01;
   "EV-51" := #_w1 AND ("Data".Ev_filter_on = 12) AND #Abilita_lavaggio_BF02;
   "EV-12" := #_w1 AND ("Data".Ev_filter_on = 13) AND #Abilita_lavaggio_BF01;
   "EV-52" := #_w1 AND ("Data".Ev_filter_on = 14) AND #Abilita_lavaggio_BF02;
   "EV-13" := #_w1 AND ("Data".Ev_filter_on = 15) AND #Abilita_lavaggio_BF01;
   "EV-53" := #_w1 AND ("Data".Ev_filter_on = 16) AND #Abilita_lavaggio_BF02;
   "EV-14" := #_w1 AND ("Data".Ev_filter_on = 17) AND #Abilita_lavaggio_BF01;
   "EV-54" := #_w1 AND ("Data".Ev_filter_on = 18) AND #Abilita_lavaggio_BF02;
   "EV-15" := #_w1 AND ("Data".Ev_filter_on = 19) AND #Abilita_lavaggio_BF01;
   "EV-55" := #_w1 AND ("Data".Ev_filter_on = 20) AND #Abilita_lavaggio_BF02;
END_REGION

REGION Network 11: wash filter
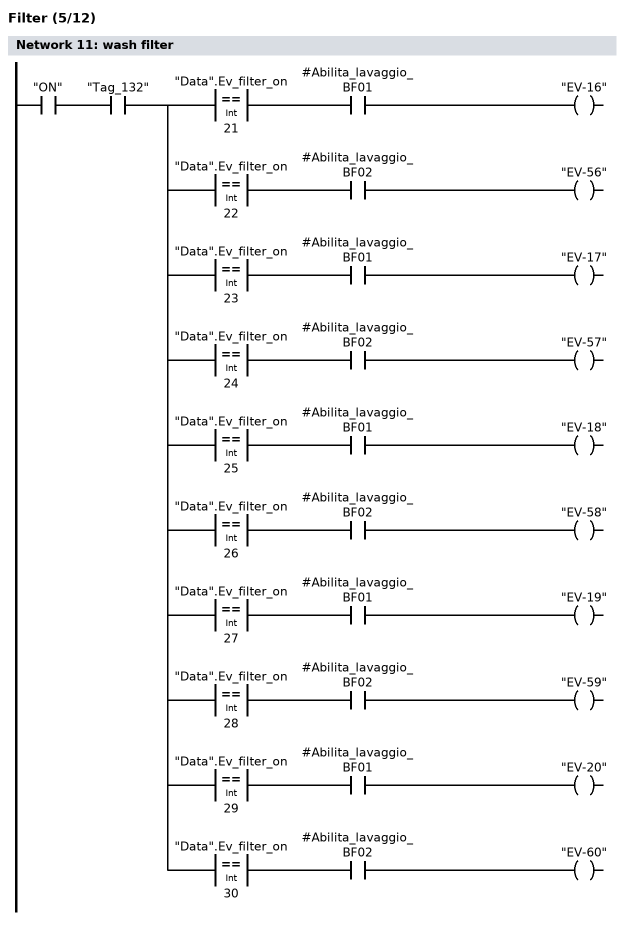
   RUNG wire#powerrail
      Contact( "ON" )
      Contact( "Tag_132" )
      wire#w1
      { S7_Templates := "SrcType := Int" } EQ_Contact(in1 := "Data".Ev_filter_on, in2 := 21)
      Contact( #Abilita_lavaggio_BF01 )
      Coil( "EV-16" )
   END_RUNG
   RUNG wire#w1
      { S7_Templates := "SrcType := Int" } EQ_Contact(in1 := "Data".Ev_filter_on, in2 := 22)
      Contact( #Abilita_lavaggio_BF02 )
      Coil( "EV-56" )
   END_RUNG
   RUNG wire#w1
      { S7_Templates := "SrcType := Int" } EQ_Contact(in1 := "Data".Ev_filter_on, in2 := 23)
      Contact( #Abilita_lavaggio_BF01 )
      Coil( "EV-17" )
   END_RUNG
   RUNG wire#w1
      { S7_Templates := "SrcType := Int" } EQ_Contact(in1 := "Data".Ev_filter_on, in2 := 24)
      Contact( #Abilita_lavaggio_BF02 )
      Coil( "EV-57" )
   END_RUNG
   RUNG wire#w1
      { S7_Templates := "SrcType := Int" } EQ_Contact(in1 := "Data".Ev_filter_on, in2 := 25)
      Contact( #Abilita_lavaggio_BF01 )
      Coil( "EV-18" )
   END_RUNG
   RUNG wire#w1
      { S7_Templates := "SrcType := Int" } EQ_Contact(in1 := "Data".Ev_filter_on, in2 := 26)
      Contact( #Abilita_lavaggio_BF02 )
      Coil( "EV-58" )
   END_RUNG
   RUNG wire#w1
      { S7_Templates := "SrcType := Int" } EQ_Contact(in1 := "Data".Ev_filter_on, in2 := 27)
      Contact( #Abilita_lavaggio_BF01 )
      Coil( "EV-19" )
   END_RUNG
   RUNG wire#w1
      { S7_Templates := "SrcType := Int" } EQ_Contact(in1 := "Data".Ev_filter_on, in2 := 28)
      Contact( #Abilita_lavaggio_BF02 )
      Coil( "EV-59" )
   END_RUNG
   RUNG wire#w1
      { S7_Templates := "SrcType := Int" } EQ_Contact(in1 := "Data".Ev_filter_on, in2 := 29)
      Contact( #Abilita_lavaggio_BF01 )
      Coil( "EV-20" )
   END_RUNG
   RUNG wire#w1
      { S7_Templates := "SrcType := Int" } EQ_Contact(in1 := "Data".Ev_filter_on, in2 := 30)
      Contact( #Abilita_lavaggio_BF02 )
      Coil( "EV-60" )
   END_RUNG
   // the same network as SCL:
   #_w1 := "ON" AND "Tag_132";
   "EV-16" := #_w1 AND ("Data".Ev_filter_on = 21) AND #Abilita_lavaggio_BF01;
   "EV-56" := #_w1 AND ("Data".Ev_filter_on = 22) AND #Abilita_lavaggio_BF02;
   "EV-17" := #_w1 AND ("Data".Ev_filter_on = 23) AND #Abilita_lavaggio_BF01;
   "EV-57" := #_w1 AND ("Data".Ev_filter_on = 24) AND #Abilita_lavaggio_BF02;
   "EV-18" := #_w1 AND ("Data".Ev_filter_on = 25) AND #Abilita_lavaggio_BF01;
   "EV-58" := #_w1 AND ("Data".Ev_filter_on = 26) AND #Abilita_lavaggio_BF02;
   "EV-19" := #_w1 AND ("Data".Ev_filter_on = 27) AND #Abilita_lavaggio_BF01;
   "EV-59" := #_w1 AND ("Data".Ev_filter_on = 28) AND #Abilita_lavaggio_BF02;
   "EV-20" := #_w1 AND ("Data".Ev_filter_on = 29) AND #Abilita_lavaggio_BF01;
   "EV-60" := #_w1 AND ("Data".Ev_filter_on = 30) AND #Abilita_lavaggio_BF02;
END_REGION

REGION Network 12: wash filter
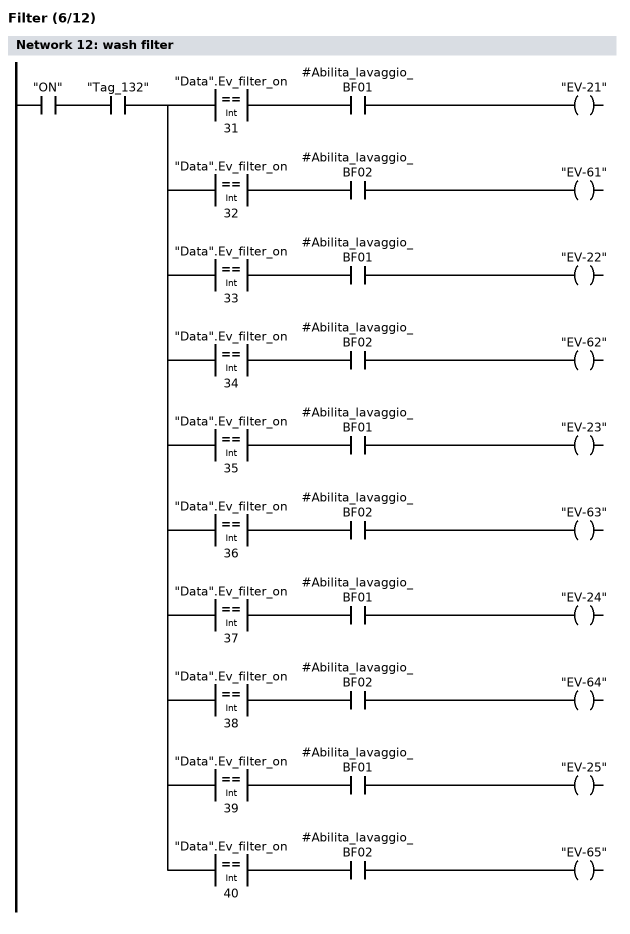
   RUNG wire#powerrail
      Contact( "ON" )
      Contact( "Tag_132" )
      wire#w1
      { S7_Templates := "SrcType := Int" } EQ_Contact(in1 := "Data".Ev_filter_on, in2 := 31)
      Contact( #Abilita_lavaggio_BF01 )
      Coil( "EV-21" )
   END_RUNG
   RUNG wire#w1
      { S7_Templates := "SrcType := Int" } EQ_Contact(in1 := "Data".Ev_filter_on, in2 := 32)
      Contact( #Abilita_lavaggio_BF02 )
      Coil( "EV-61" )
   END_RUNG
   RUNG wire#w1
      { S7_Templates := "SrcType := Int" } EQ_Contact(in1 := "Data".Ev_filter_on, in2 := 33)
      Contact( #Abilita_lavaggio_BF01 )
      Coil( "EV-22" )
   END_RUNG
   RUNG wire#w1
      { S7_Templates := "SrcType := Int" } EQ_Contact(in1 := "Data".Ev_filter_on, in2 := 34)
      Contact( #Abilita_lavaggio_BF02 )
      Coil( "EV-62" )
   END_RUNG
   RUNG wire#w1
      { S7_Templates := "SrcType := Int" } EQ_Contact(in1 := "Data".Ev_filter_on, in2 := 35)
      Contact( #Abilita_lavaggio_BF01 )
      Coil( "EV-23" )
   END_RUNG
   RUNG wire#w1
      { S7_Templates := "SrcType := Int" } EQ_Contact(in1 := "Data".Ev_filter_on, in2 := 36)
      Contact( #Abilita_lavaggio_BF02 )
      Coil( "EV-63" )
   END_RUNG
   RUNG wire#w1
      { S7_Templates := "SrcType := Int" } EQ_Contact(in1 := "Data".Ev_filter_on, in2 := 37)
      Contact( #Abilita_lavaggio_BF01 )
      Coil( "EV-24" )
   END_RUNG
   RUNG wire#w1
      { S7_Templates := "SrcType := Int" } EQ_Contact(in1 := "Data".Ev_filter_on, in2 := 38)
      Contact( #Abilita_lavaggio_BF02 )
      Coil( "EV-64" )
   END_RUNG
   RUNG wire#w1
      { S7_Templates := "SrcType := Int" } EQ_Contact(in1 := "Data".Ev_filter_on, in2 := 39)
      Contact( #Abilita_lavaggio_BF01 )
      Coil( "EV-25" )
   END_RUNG
   RUNG wire#w1
      { S7_Templates := "SrcType := Int" } EQ_Contact(in1 := "Data".Ev_filter_on, in2 := 40)
      Contact( #Abilita_lavaggio_BF02 )
      Coil( "EV-65" )
   END_RUNG
   // the same network as SCL:
   #_w1 := "ON" AND "Tag_132";
   "EV-21" := #_w1 AND ("Data".Ev_filter_on = 31) AND #Abilita_lavaggio_BF01;
   "EV-61" := #_w1 AND ("Data".Ev_filter_on = 32) AND #Abilita_lavaggio_BF02;
   "EV-22" := #_w1 AND ("Data".Ev_filter_on = 33) AND #Abilita_lavaggio_BF01;
   "EV-62" := #_w1 AND ("Data".Ev_filter_on = 34) AND #Abilita_lavaggio_BF02;
   "EV-23" := #_w1 AND ("Data".Ev_filter_on = 35) AND #Abilita_lavaggio_BF01;
   "EV-63" := #_w1 AND ("Data".Ev_filter_on = 36) AND #Abilita_lavaggio_BF02;
   "EV-24" := #_w1 AND ("Data".Ev_filter_on = 37) AND #Abilita_lavaggio_BF01;
   "EV-64" := #_w1 AND ("Data".Ev_filter_on = 38) AND #Abilita_lavaggio_BF02;
   "EV-25" := #_w1 AND ("Data".Ev_filter_on = 39) AND #Abilita_lavaggio_BF01;
   "EV-65" := #_w1 AND ("Data".Ev_filter_on = 40) AND #Abilita_lavaggio_BF02;
END_REGION

REGION Network 13: wash filter
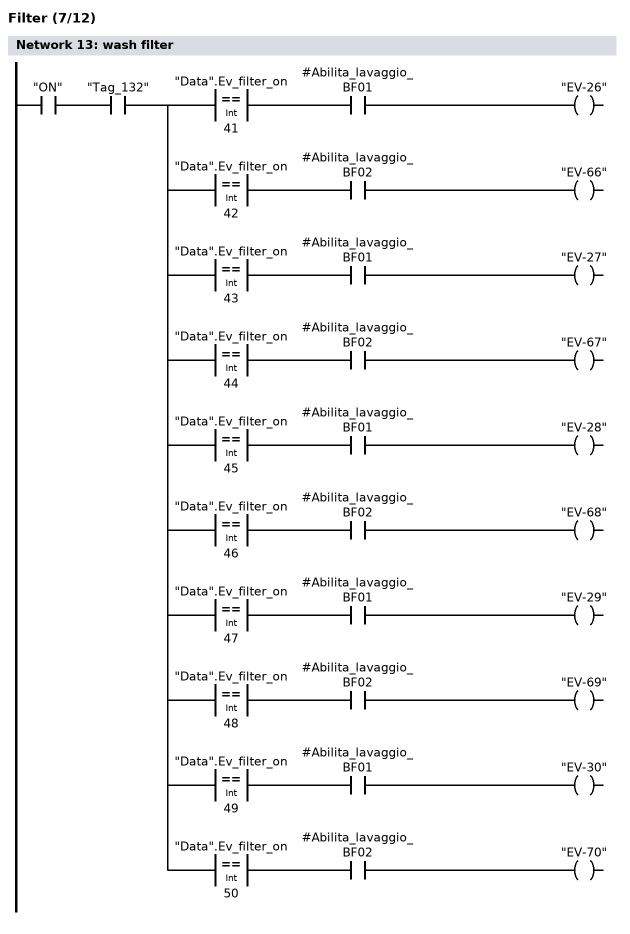
   RUNG wire#powerrail
      Contact( "ON" )
      Contact( "Tag_132" )
      wire#w1
      { S7_Templates := "SrcType := Int" } EQ_Contact(in1 := "Data".Ev_filter_on, in2 := 41)
      Contact( #Abilita_lavaggio_BF01 )
      Coil( "EV-26" )
   END_RUNG
   RUNG wire#w1
      { S7_Templates := "SrcType := Int" } EQ_Contact(in1 := "Data".Ev_filter_on, in2 := 42)
      Contact( #Abilita_lavaggio_BF02 )
      Coil( "EV-66" )
   END_RUNG
   RUNG wire#w1
      { S7_Templates := "SrcType := Int" } EQ_Contact(in1 := "Data".Ev_filter_on, in2 := 43)
      Contact( #Abilita_lavaggio_BF01 )
      Coil( "EV-27" )
   END_RUNG
   RUNG wire#w1
      { S7_Templates := "SrcType := Int" } EQ_Contact(in1 := "Data".Ev_filter_on, in2 := 44)
      Contact( #Abilita_lavaggio_BF02 )
      Coil( "EV-67" )
   END_RUNG
   RUNG wire#w1
      { S7_Templates := "SrcType := Int" } EQ_Contact(in1 := "Data".Ev_filter_on, in2 := 45)
      Contact( #Abilita_lavaggio_BF01 )
      Coil( "EV-28" )
   END_RUNG
   RUNG wire#w1
      { S7_Templates := "SrcType := Int" } EQ_Contact(in1 := "Data".Ev_filter_on, in2 := 46)
      Contact( #Abilita_lavaggio_BF02 )
      Coil( "EV-68" )
   END_RUNG
   RUNG wire#w1
      { S7_Templates := "SrcType := Int" } EQ_Contact(in1 := "Data".Ev_filter_on, in2 := 47)
      Contact( #Abilita_lavaggio_BF01 )
      Coil( "EV-29" )
   END_RUNG
   RUNG wire#w1
      { S7_Templates := "SrcType := Int" } EQ_Contact(in1 := "Data".Ev_filter_on, in2 := 48)
      Contact( #Abilita_lavaggio_BF02 )
      Coil( "EV-69" )
   END_RUNG
   RUNG wire#w1
      { S7_Templates := "SrcType := Int" } EQ_Contact(in1 := "Data".Ev_filter_on, in2 := 49)
      Contact( #Abilita_lavaggio_BF01 )
      Coil( "EV-30" )
   END_RUNG
   RUNG wire#w1
      { S7_Templates := "SrcType := Int" } EQ_Contact(in1 := "Data".Ev_filter_on, in2 := 50)
      Contact( #Abilita_lavaggio_BF02 )
      Coil( "EV-70" )
   END_RUNG
   // the same network as SCL:
   #_w1 := "ON" AND "Tag_132";
   "EV-26" := #_w1 AND ("Data".Ev_filter_on = 41) AND #Abilita_lavaggio_BF01;
   "EV-66" := #_w1 AND ("Data".Ev_filter_on = 42) AND #Abilita_lavaggio_BF02;
   "EV-27" := #_w1 AND ("Data".Ev_filter_on = 43) AND #Abilita_lavaggio_BF01;
   "EV-67" := #_w1 AND ("Data".Ev_filter_on = 44) AND #Abilita_lavaggio_BF02;
   "EV-28" := #_w1 AND ("Data".Ev_filter_on = 45) AND #Abilita_lavaggio_BF01;
   "EV-68" := #_w1 AND ("Data".Ev_filter_on = 46) AND #Abilita_lavaggio_BF02;
   "EV-29" := #_w1 AND ("Data".Ev_filter_on = 47) AND #Abilita_lavaggio_BF01;
   "EV-69" := #_w1 AND ("Data".Ev_filter_on = 48) AND #Abilita_lavaggio_BF02;
   "EV-30" := #_w1 AND ("Data".Ev_filter_on = 49) AND #Abilita_lavaggio_BF01;
   "EV-70" := #_w1 AND ("Data".Ev_filter_on = 50) AND #Abilita_lavaggio_BF02;
END_REGION

REGION Network 14: wash filter
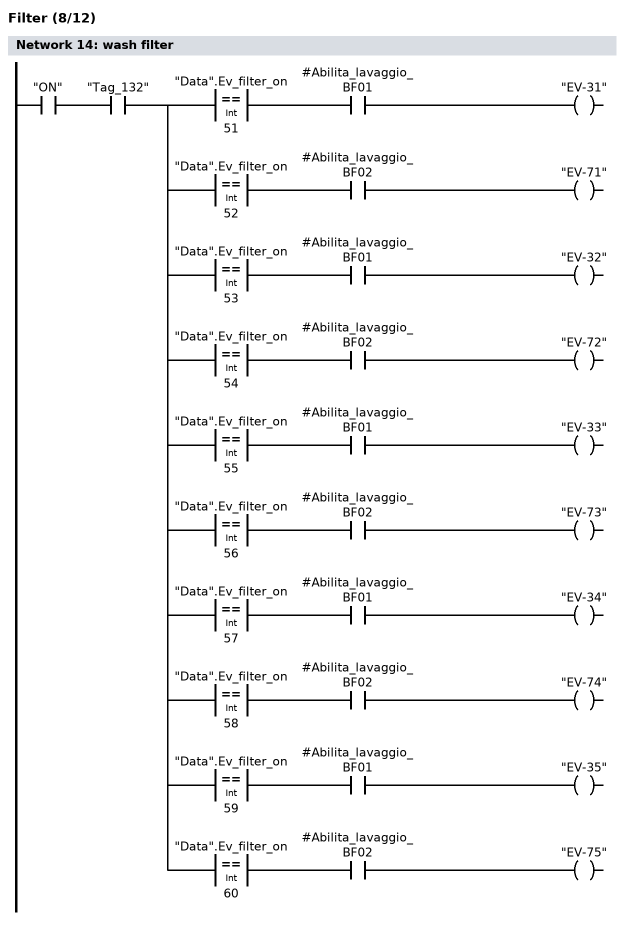
   RUNG wire#powerrail
      Contact( "ON" )
      Contact( "Tag_132" )
      wire#w1
      { S7_Templates := "SrcType := Int" } EQ_Contact(in1 := "Data".Ev_filter_on, in2 := 51)
      Contact( #Abilita_lavaggio_BF01 )
      Coil( "EV-31" )
   END_RUNG
   RUNG wire#w1
      { S7_Templates := "SrcType := Int" } EQ_Contact(in1 := "Data".Ev_filter_on, in2 := 52)
      Contact( #Abilita_lavaggio_BF02 )
      Coil( "EV-71" )
   END_RUNG
   RUNG wire#w1
      { S7_Templates := "SrcType := Int" } EQ_Contact(in1 := "Data".Ev_filter_on, in2 := 53)
      Contact( #Abilita_lavaggio_BF01 )
      Coil( "EV-32" )
   END_RUNG
   RUNG wire#w1
      { S7_Templates := "SrcType := Int" } EQ_Contact(in1 := "Data".Ev_filter_on, in2 := 54)
      Contact( #Abilita_lavaggio_BF02 )
      Coil( "EV-72" )
   END_RUNG
   RUNG wire#w1
      { S7_Templates := "SrcType := Int" } EQ_Contact(in1 := "Data".Ev_filter_on, in2 := 55)
      Contact( #Abilita_lavaggio_BF01 )
      Coil( "EV-33" )
   END_RUNG
   RUNG wire#w1
      { S7_Templates := "SrcType := Int" } EQ_Contact(in1 := "Data".Ev_filter_on, in2 := 56)
      Contact( #Abilita_lavaggio_BF02 )
      Coil( "EV-73" )
   END_RUNG
   RUNG wire#w1
      { S7_Templates := "SrcType := Int" } EQ_Contact(in1 := "Data".Ev_filter_on, in2 := 57)
      Contact( #Abilita_lavaggio_BF01 )
      Coil( "EV-34" )
   END_RUNG
   RUNG wire#w1
      { S7_Templates := "SrcType := Int" } EQ_Contact(in1 := "Data".Ev_filter_on, in2 := 58)
      Contact( #Abilita_lavaggio_BF02 )
      Coil( "EV-74" )
   END_RUNG
   RUNG wire#w1
      { S7_Templates := "SrcType := Int" } EQ_Contact(in1 := "Data".Ev_filter_on, in2 := 59)
      Contact( #Abilita_lavaggio_BF01 )
      Coil( "EV-35" )
   END_RUNG
   RUNG wire#w1
      { S7_Templates := "SrcType := Int" } EQ_Contact(in1 := "Data".Ev_filter_on, in2 := 60)
      Contact( #Abilita_lavaggio_BF02 )
      Coil( "EV-75" )
   END_RUNG
   // the same network as SCL:
   #_w1 := "ON" AND "Tag_132";
   "EV-31" := #_w1 AND ("Data".Ev_filter_on = 51) AND #Abilita_lavaggio_BF01;
   "EV-71" := #_w1 AND ("Data".Ev_filter_on = 52) AND #Abilita_lavaggio_BF02;
   "EV-32" := #_w1 AND ("Data".Ev_filter_on = 53) AND #Abilita_lavaggio_BF01;
   "EV-72" := #_w1 AND ("Data".Ev_filter_on = 54) AND #Abilita_lavaggio_BF02;
   "EV-33" := #_w1 AND ("Data".Ev_filter_on = 55) AND #Abilita_lavaggio_BF01;
   "EV-73" := #_w1 AND ("Data".Ev_filter_on = 56) AND #Abilita_lavaggio_BF02;
   "EV-34" := #_w1 AND ("Data".Ev_filter_on = 57) AND #Abilita_lavaggio_BF01;
   "EV-74" := #_w1 AND ("Data".Ev_filter_on = 58) AND #Abilita_lavaggio_BF02;
   "EV-35" := #_w1 AND ("Data".Ev_filter_on = 59) AND #Abilita_lavaggio_BF01;
   "EV-75" := #_w1 AND ("Data".Ev_filter_on = 60) AND #Abilita_lavaggio_BF02;
END_REGION

REGION Network 15: wash filter
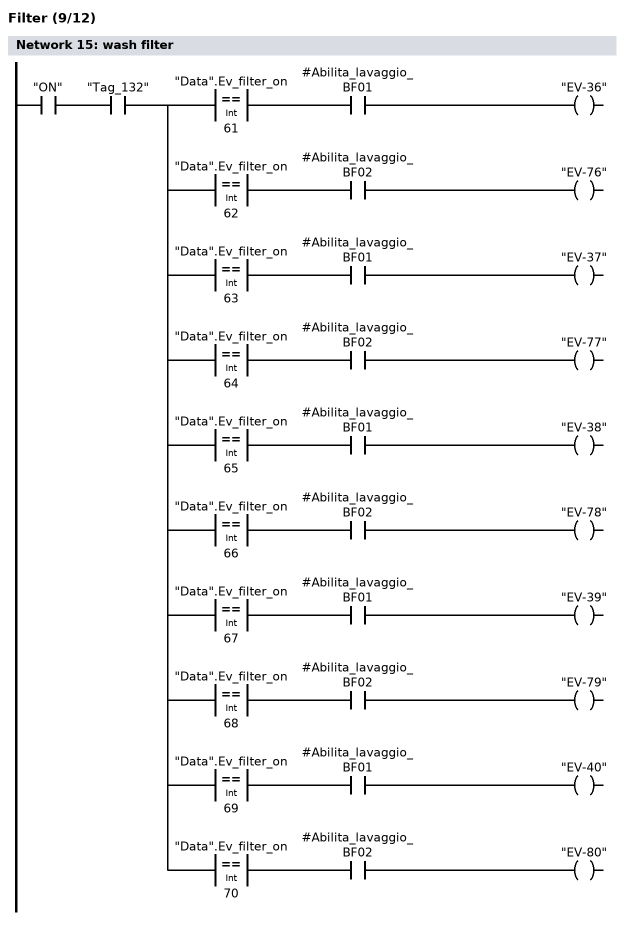
   RUNG wire#powerrail
      Contact( "ON" )
      Contact( "Tag_132" )
      wire#w1
      { S7_Templates := "SrcType := Int" } EQ_Contact(in1 := "Data".Ev_filter_on, in2 := 61)
      Contact( #Abilita_lavaggio_BF01 )
      Coil( "EV-36" )
   END_RUNG
   RUNG wire#w1
      { S7_Templates := "SrcType := Int" } EQ_Contact(in1 := "Data".Ev_filter_on, in2 := 62)
      Contact( #Abilita_lavaggio_BF02 )
      Coil( "EV-76" )
   END_RUNG
   RUNG wire#w1
      { S7_Templates := "SrcType := Int" } EQ_Contact(in1 := "Data".Ev_filter_on, in2 := 63)
      Contact( #Abilita_lavaggio_BF01 )
      Coil( "EV-37" )
   END_RUNG
   RUNG wire#w1
      { S7_Templates := "SrcType := Int" } EQ_Contact(in1 := "Data".Ev_filter_on, in2 := 64)
      Contact( #Abilita_lavaggio_BF02 )
      Coil( "EV-77" )
   END_RUNG
   RUNG wire#w1
      { S7_Templates := "SrcType := Int" } EQ_Contact(in1 := "Data".Ev_filter_on, in2 := 65)
      Contact( #Abilita_lavaggio_BF01 )
      Coil( "EV-38" )
   END_RUNG
   RUNG wire#w1
      { S7_Templates := "SrcType := Int" } EQ_Contact(in1 := "Data".Ev_filter_on, in2 := 66)
      Contact( #Abilita_lavaggio_BF02 )
      Coil( "EV-78" )
   END_RUNG
   RUNG wire#w1
      { S7_Templates := "SrcType := Int" } EQ_Contact(in1 := "Data".Ev_filter_on, in2 := 67)
      Contact( #Abilita_lavaggio_BF01 )
      Coil( "EV-39" )
   END_RUNG
   RUNG wire#w1
      { S7_Templates := "SrcType := Int" } EQ_Contact(in1 := "Data".Ev_filter_on, in2 := 68)
      Contact( #Abilita_lavaggio_BF02 )
      Coil( "EV-79" )
   END_RUNG
   RUNG wire#w1
      { S7_Templates := "SrcType := Int" } EQ_Contact(in1 := "Data".Ev_filter_on, in2 := 69)
      Contact( #Abilita_lavaggio_BF01 )
      Coil( "EV-40" )
   END_RUNG
   RUNG wire#w1
      { S7_Templates := "SrcType := Int" } EQ_Contact(in1 := "Data".Ev_filter_on, in2 := 70)
      Contact( #Abilita_lavaggio_BF02 )
      Coil( "EV-80" )
   END_RUNG
   // the same network as SCL:
   #_w1 := "ON" AND "Tag_132";
   "EV-36" := #_w1 AND ("Data".Ev_filter_on = 61) AND #Abilita_lavaggio_BF01;
   "EV-76" := #_w1 AND ("Data".Ev_filter_on = 62) AND #Abilita_lavaggio_BF02;
   "EV-37" := #_w1 AND ("Data".Ev_filter_on = 63) AND #Abilita_lavaggio_BF01;
   "EV-77" := #_w1 AND ("Data".Ev_filter_on = 64) AND #Abilita_lavaggio_BF02;
   "EV-38" := #_w1 AND ("Data".Ev_filter_on = 65) AND #Abilita_lavaggio_BF01;
   "EV-78" := #_w1 AND ("Data".Ev_filter_on = 66) AND #Abilita_lavaggio_BF02;
   "EV-39" := #_w1 AND ("Data".Ev_filter_on = 67) AND #Abilita_lavaggio_BF01;
   "EV-79" := #_w1 AND ("Data".Ev_filter_on = 68) AND #Abilita_lavaggio_BF02;
   "EV-40" := #_w1 AND ("Data".Ev_filter_on = 69) AND #Abilita_lavaggio_BF01;
   "EV-80" := #_w1 AND ("Data".Ev_filter_on = 70) AND #Abilita_lavaggio_BF02;
END_REGION

REGION Network 16: wash filter
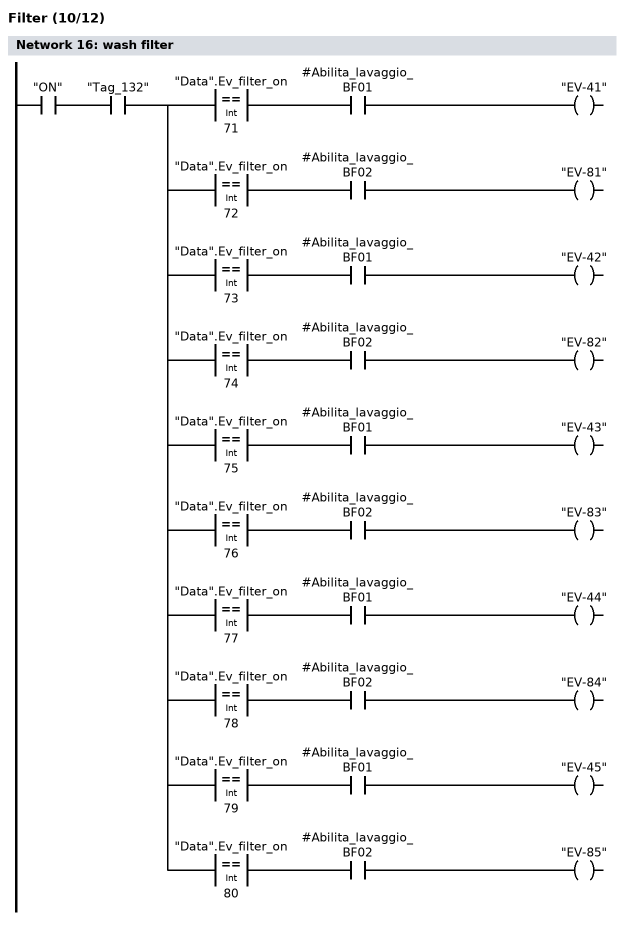
   RUNG wire#powerrail
      Contact( "ON" )
      Contact( "Tag_132" )
      wire#w1
      { S7_Templates := "SrcType := Int" } EQ_Contact(in1 := "Data".Ev_filter_on, in2 := 71)
      Contact( #Abilita_lavaggio_BF01 )
      Coil( "EV-41" )
   END_RUNG
   RUNG wire#w1
      { S7_Templates := "SrcType := Int" } EQ_Contact(in1 := "Data".Ev_filter_on, in2 := 72)
      Contact( #Abilita_lavaggio_BF02 )
      Coil( "EV-81" )
   END_RUNG
   RUNG wire#w1
      { S7_Templates := "SrcType := Int" } EQ_Contact(in1 := "Data".Ev_filter_on, in2 := 73)
      Contact( #Abilita_lavaggio_BF01 )
      Coil( "EV-42" )
   END_RUNG
   RUNG wire#w1
      { S7_Templates := "SrcType := Int" } EQ_Contact(in1 := "Data".Ev_filter_on, in2 := 74)
      Contact( #Abilita_lavaggio_BF02 )
      Coil( "EV-82" )
   END_RUNG
   RUNG wire#w1
      { S7_Templates := "SrcType := Int" } EQ_Contact(in1 := "Data".Ev_filter_on, in2 := 75)
      Contact( #Abilita_lavaggio_BF01 )
      Coil( "EV-43" )
   END_RUNG
   RUNG wire#w1
      { S7_Templates := "SrcType := Int" } EQ_Contact(in1 := "Data".Ev_filter_on, in2 := 76)
      Contact( #Abilita_lavaggio_BF02 )
      Coil( "EV-83" )
   END_RUNG
   RUNG wire#w1
      { S7_Templates := "SrcType := Int" } EQ_Contact(in1 := "Data".Ev_filter_on, in2 := 77)
      Contact( #Abilita_lavaggio_BF01 )
      Coil( "EV-44" )
   END_RUNG
   RUNG wire#w1
      { S7_Templates := "SrcType := Int" } EQ_Contact(in1 := "Data".Ev_filter_on, in2 := 78)
      Contact( #Abilita_lavaggio_BF02 )
      Coil( "EV-84" )
   END_RUNG
   RUNG wire#w1
      { S7_Templates := "SrcType := Int" } EQ_Contact(in1 := "Data".Ev_filter_on, in2 := 79)
      Contact( #Abilita_lavaggio_BF01 )
      Coil( "EV-45" )
   END_RUNG
   RUNG wire#w1
      { S7_Templates := "SrcType := Int" } EQ_Contact(in1 := "Data".Ev_filter_on, in2 := 80)
      Contact( #Abilita_lavaggio_BF02 )
      Coil( "EV-85" )
   END_RUNG
   // the same network as SCL:
   #_w1 := "ON" AND "Tag_132";
   "EV-41" := #_w1 AND ("Data".Ev_filter_on = 71) AND #Abilita_lavaggio_BF01;
   "EV-81" := #_w1 AND ("Data".Ev_filter_on = 72) AND #Abilita_lavaggio_BF02;
   "EV-42" := #_w1 AND ("Data".Ev_filter_on = 73) AND #Abilita_lavaggio_BF01;
   "EV-82" := #_w1 AND ("Data".Ev_filter_on = 74) AND #Abilita_lavaggio_BF02;
   "EV-43" := #_w1 AND ("Data".Ev_filter_on = 75) AND #Abilita_lavaggio_BF01;
   "EV-83" := #_w1 AND ("Data".Ev_filter_on = 76) AND #Abilita_lavaggio_BF02;
   "EV-44" := #_w1 AND ("Data".Ev_filter_on = 77) AND #Abilita_lavaggio_BF01;
   "EV-84" := #_w1 AND ("Data".Ev_filter_on = 78) AND #Abilita_lavaggio_BF02;
   "EV-45" := #_w1 AND ("Data".Ev_filter_on = 79) AND #Abilita_lavaggio_BF01;
   "EV-85" := #_w1 AND ("Data".Ev_filter_on = 80) AND #Abilita_lavaggio_BF02;
END_REGION

REGION Network 17: wash filter
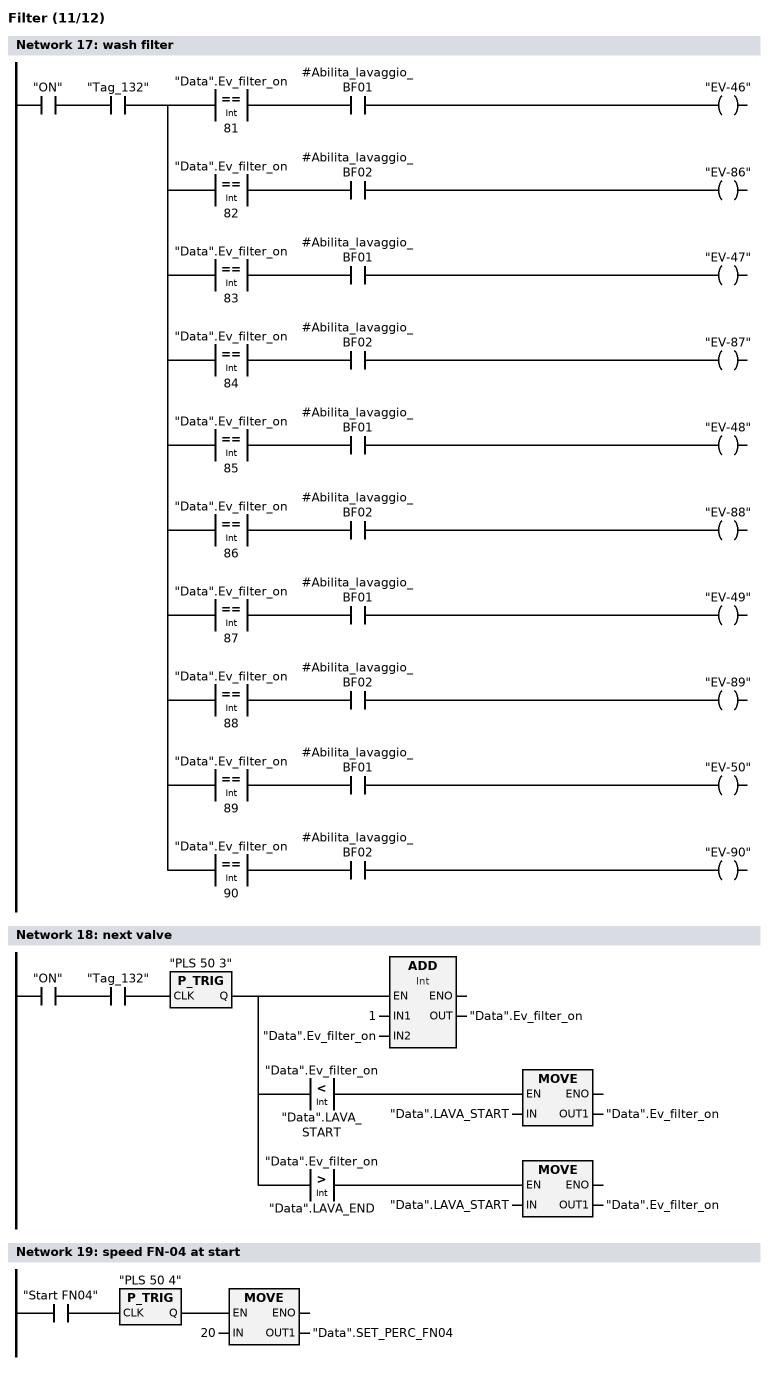
   RUNG wire#powerrail
      Contact( "ON" )
      Contact( "Tag_132" )
      wire#w1
      { S7_Templates := "SrcType := Int" } EQ_Contact(in1 := "Data".Ev_filter_on, in2 := 81)
      Contact( #Abilita_lavaggio_BF01 )
      Coil( "EV-46" )
   END_RUNG
   RUNG wire#w1
      { S7_Templates := "SrcType := Int" } EQ_Contact(in1 := "Data".Ev_filter_on, in2 := 82)
      Contact( #Abilita_lavaggio_BF02 )
      Coil( "EV-86" )
   END_RUNG
   RUNG wire#w1
      { S7_Templates := "SrcType := Int" } EQ_Contact(in1 := "Data".Ev_filter_on, in2 := 83)
      Contact( #Abilita_lavaggio_BF01 )
      Coil( "EV-47" )
   END_RUNG
   RUNG wire#w1
      { S7_Templates := "SrcType := Int" } EQ_Contact(in1 := "Data".Ev_filter_on, in2 := 84)
      Contact( #Abilita_lavaggio_BF02 )
      Coil( "EV-87" )
   END_RUNG
   RUNG wire#w1
      { S7_Templates := "SrcType := Int" } EQ_Contact(in1 := "Data".Ev_filter_on, in2 := 85)
      Contact( #Abilita_lavaggio_BF01 )
      Coil( "EV-48" )
   END_RUNG
   RUNG wire#w1
      { S7_Templates := "SrcType := Int" } EQ_Contact(in1 := "Data".Ev_filter_on, in2 := 86)
      Contact( #Abilita_lavaggio_BF02 )
      Coil( "EV-88" )
   END_RUNG
   RUNG wire#w1
      { S7_Templates := "SrcType := Int" } EQ_Contact(in1 := "Data".Ev_filter_on, in2 := 87)
      Contact( #Abilita_lavaggio_BF01 )
      Coil( "EV-49" )
   END_RUNG
   RUNG wire#w1
      { S7_Templates := "SrcType := Int" } EQ_Contact(in1 := "Data".Ev_filter_on, in2 := 88)
      Contact( #Abilita_lavaggio_BF02 )
      Coil( "EV-89" )
   END_RUNG
   RUNG wire#w1
      { S7_Templates := "SrcType := Int" } EQ_Contact(in1 := "Data".Ev_filter_on, in2 := 89)
      Contact( #Abilita_lavaggio_BF01 )
      Coil( "EV-50" )
   END_RUNG
   RUNG wire#w1
      { S7_Templates := "SrcType := Int" } EQ_Contact(in1 := "Data".Ev_filter_on, in2 := 90)
      Contact( #Abilita_lavaggio_BF02 )
      Coil( "EV-90" )
   END_RUNG
   // the same network as SCL:
   #_w1 := "ON" AND "Tag_132";
   "EV-46" := #_w1 AND ("Data".Ev_filter_on = 81) AND #Abilita_lavaggio_BF01;
   "EV-86" := #_w1 AND ("Data".Ev_filter_on = 82) AND #Abilita_lavaggio_BF02;
   "EV-47" := #_w1 AND ("Data".Ev_filter_on = 83) AND #Abilita_lavaggio_BF01;
   "EV-87" := #_w1 AND ("Data".Ev_filter_on = 84) AND #Abilita_lavaggio_BF02;
   "EV-48" := #_w1 AND ("Data".Ev_filter_on = 85) AND #Abilita_lavaggio_BF01;
   "EV-88" := #_w1 AND ("Data".Ev_filter_on = 86) AND #Abilita_lavaggio_BF02;
   "EV-49" := #_w1 AND ("Data".Ev_filter_on = 87) AND #Abilita_lavaggio_BF01;
   "EV-89" := #_w1 AND ("Data".Ev_filter_on = 88) AND #Abilita_lavaggio_BF02;
   "EV-50" := #_w1 AND ("Data".Ev_filter_on = 89) AND #Abilita_lavaggio_BF01;
   "EV-90" := #_w1 AND ("Data".Ev_filter_on = 90) AND #Abilita_lavaggio_BF02;
END_REGION

REGION Network 18: next valve
   RUNG wire#powerrail
      Contact( "ON" )
      Contact( "Tag_132" )
      P_Trig( "PLS 50 3" )
      wire#w1
      { S7_Templates := "SrcType := Int"; S7_GenerateENO := "TRUE" } Add(in1 := 1, in2 := "Data".Ev_filter_on, out => "Data".Ev_filter_on)
   END_RUNG
   RUNG wire#w1
      { S7_Templates := "SrcType := Int" } LT_Contact(in1 := "Data".Ev_filter_on, in2 := "Data".LAVA_START)
      { S7_GenerateENO := "TRUE" } Move(in := "Data".LAVA_START, out1 => "Data".Ev_filter_on)
   END_RUNG
   RUNG wire#w1
      { S7_Templates := "SrcType := Int" } GT_Contact(in1 := "Data".Ev_filter_on, in2 := "Data".LAVA_END)
      { S7_GenerateENO := "TRUE" } Move(in := "Data".LAVA_START, out1 => "Data".Ev_filter_on)
   END_RUNG
   // the same network as SCL:
   #_w1 := "ON" AND "Tag_132";
   #_w2 := #_w1 AND NOT "PLS 50 3";   // rising edge
   "PLS 50 3" := #_w1;
   IF #_w2 THEN "Data".Ev_filter_on := 1 + "Data".Ev_filter_on; END_IF;
   IF #_w2 AND ("Data".Ev_filter_on < "Data".LAVA_START) THEN
       "Data".Ev_filter_on := "Data".LAVA_START;
   END_IF;
   IF #_w2 AND ("Data".Ev_filter_on > "Data".LAVA_END) THEN "Data".Ev_filter_on := "Data".LAVA_START; END_IF;
END_REGION

REGION Network 19: speed FN-04 at start
   RUNG wire#powerrail
      Contact( "Start FN04" )
      P_Trig( "PLS 50 4" )
      { S7_GenerateENO := "TRUE" } Move(in := 20, out1 => "Data".SET_PERC_FN04)
   END_RUNG
   // the same network as SCL:
   #_w1 := "Start FN04" AND NOT "PLS 50 4";   // rising edge
   "PLS 50 4" := "Start FN04";
   IF #_w1 THEN "Data".SET_PERC_FN04 := 20; END_IF;
END_REGION

REGION Network 20: DP-01 Control loop
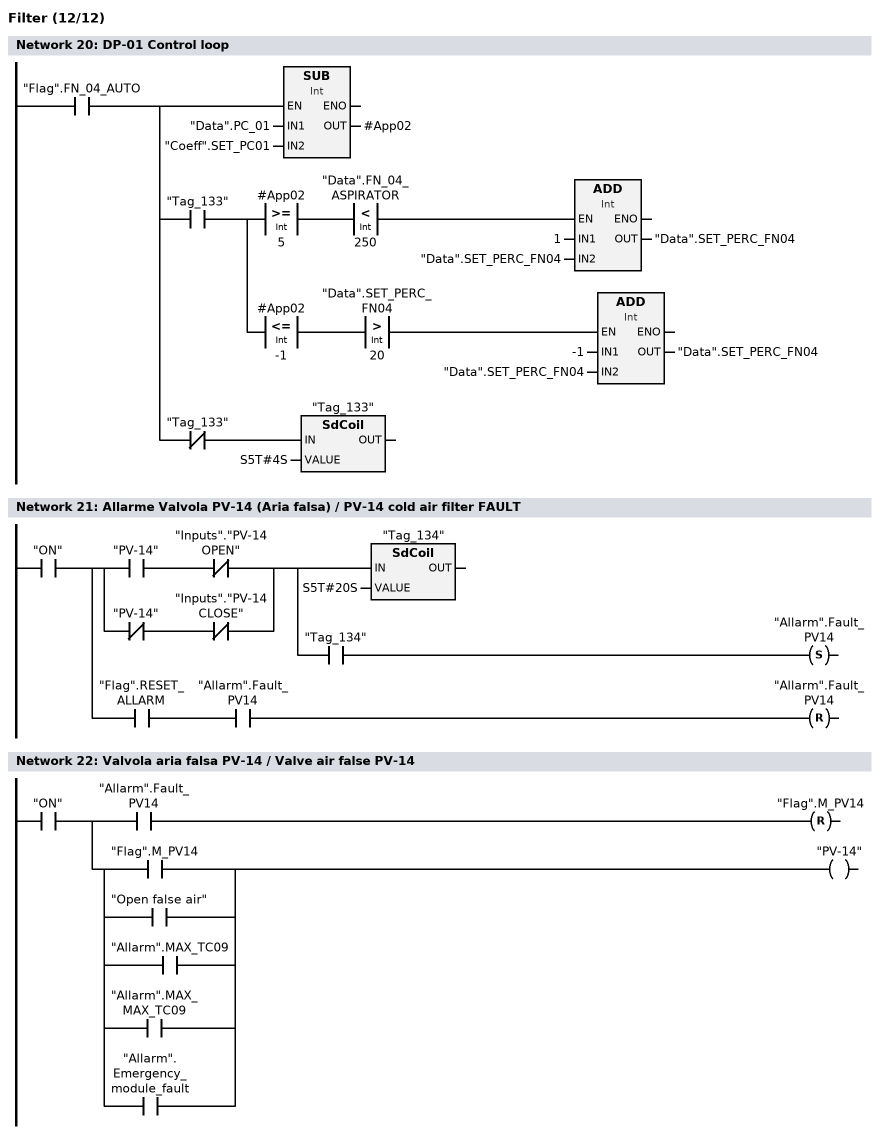
   // no SCL statement known for SdCoil: written as a call
   IF "Flag".FN_04_AUTO THEN #App02 := "Data".PC_01 - "Coeff".SET_PC01; END_IF;
   #_w1 := "Flag".FN_04_AUTO AND "Tag_133";
   IF #_w1 AND (#App02 >= 5) AND ("Data".FN_04_ASPIRATOR < 250) THEN
       "Data".SET_PERC_FN04 := 1 + "Data".SET_PERC_FN04;
   END_IF;
   IF #_w1 AND (#App02 <= (-1)) AND ("Data".SET_PERC_FN04 > 20) THEN
       "Data".SET_PERC_FN04 := (-1) + "Data".SET_PERC_FN04;
   END_IF;
   SdCoil(in := "Flag".FN_04_AUTO AND NOT "Tag_133", value := S5T#4S, operand := "Tag_133");
END_REGION

REGION Network 21: Allarme Valvola PV-14 (Aria falsa) / PV-14 cold air filter FAULT
   // no SCL statement known for SdCoil: written as a call
   #_w1 := "ON" AND (("PV-14" AND NOT "Inputs"."PV-14 OPEN") OR (NOT "PV-14" AND NOT "Inputs"."PV-14 CLOSE"));
   #_w2 := "ON";
   SdCoil(in := #_w1, value := S5T#20S, operand := "Tag_134");
   IF #_w1 AND "Tag_134" THEN "Allarm".Fault_PV14 := TRUE; END_IF;
   IF #_w2 AND "Flag".RESET_ALLARM AND "Allarm".Fault_PV14 THEN "Allarm".Fault_PV14 := FALSE; END_IF;
END_REGION

REGION Network 22: Valvola aria falsa PV-14 / Valve air false PV-14
   RUNG wire#powerrail
      Contact( "ON" )
      wire#w1
      Contact( "Allarm".Fault_PV14 )
      R_Coil( "Flag".M_PV14 )
   END_RUNG
   RUNG wire#w1
      Contact( "Flag".M_PV14 )
      wire#w2
      Coil( "PV-14" )
   END_RUNG
   RUNG wire#w1
      Contact( "Open false air" )
   END_RUNG wire#w2
   RUNG wire#w1
      Contact( "Allarm".MAX_TC09 )
   END_RUNG wire#w2
   RUNG wire#w1
      Contact( "Allarm".MAX_MAX_TC09 )
   END_RUNG wire#w2
   RUNG wire#w1
      Contact( "Allarm".Emergency_module_fault )
   END_RUNG wire#w2
   // the same network as SCL:
   IF "ON" AND "Allarm".Fault_PV14 THEN "Flag".M_PV14 := FALSE; END_IF;
   "PV-14" := "ON" AND ("Flag".M_PV14 OR "Open false air" OR "Allarm".MAX_TC09 OR "Allarm".MAX_MAX_TC09 OR "Allarm".Emergency_module_fault);
END_REGION

REGION Network 23 (SCL)
   (* IF "EV-11" OR "EV-12" OR "EV-13" OR "EV-14" OR "EV-15" OR "EV-16" OR "EV-17" OR "EV-18" OR "EV-19" OR "EV-20" OR
       "EV-21" OR "EV-22" OR "EV-23" OR "EV-24" OR "EV-25" OR "EV-26" OR "EV-27" OR "EV-28" OR "EV-29" OR "EV-30" OR
       "EV-31" OR "EV-32" OR "EV-33" OR "EV-34" OR "EV-35" OR "EV-36" OR "EV-37" OR "EV-38" OR "EV-39" OR "EV-40" OR
       "EV-41" OR "EV-42" OR "EV-43" OR "EV-44" OR "EV-45" OR "EV-46" OR "EV-47" OR "EV-48" OR "EV-49" OR "EV-50" THEN
           "BF01_RUN":=TRUE;
       ELSE 
           "BF01_RUN" := FALSE;
   END_IF;

   IF "EV-51" OR "EV-52" OR "EV-53" OR "EV-54" OR "EV-55" OR "EV-56" OR "EV-57" OR "EV-58" OR "EV-59" OR "EV-60" OR
       "EV-61" OR "EV-62" OR "EV-63" OR "EV-64" OR "EV-65" OR "EV-66" OR "EV-67" OR "EV-68" OR "EV-69" OR "EV-70" OR
       "EV-71" OR "EV-72" OR "EV-73" OR "EV-74" OR "EV-75" OR "EV-76" OR "EV-77" OR "EV-78" OR "EV-79" OR "EV-80" OR
       "EV-81" OR "EV-82" OR "EV-83" OR "EV-84" OR "EV-85" OR "EV-86" OR "EV-87" OR "EV-88" OR "EV-89" OR "EV-90" THEN
           "BF02_RUN" := TRUE;
       ELSE
           "BF02_RUN" := FALSE;
   END_IF; *)
END_REGION
END_FUNCTION

FUNCTION "Motor/Alarm Client" : Void   // FC9, LAD
TITLE = Client motoprs and alarms
{ S7_Optimized_Access := 'FALSE' }
VERSION : 0.1
BEGIN

REGION Network 1: client motor 1 Allarm / Apron conveyor fault (CL01)
